	(**)
	bDriveDiagMessageAndNumber  : BOOL;
	m_GetDriveStatusState:INT;
	GetDriveStatusStateDone:BOOL;
	GetDriveStatusStateError:BOOL;
	GetDriveStatusTON: TON;
	//	
	fb_SoEReadDiagMessage_LeftTop: FB_SoEReadDiagMessage;
	fb_SoEReadDiagMessage_RightTop: FB_SoEReadDiagMessage;
	fb_SoEReadDiagMessage_LeftBottom: FB_SoEReadDiagMessage;
	fb_SoEReadDiagMessage_RightBottom: FB_SoEReadDiagMessage;
	DriveDiagMessage_LeftTop:STRING;
	DriveDiagMessage_RightTop:STRING;
	DriveDiagMessage_LeftBottom:STRING;
	DriveDiagMessage_RightBottom:STRING;
	fb_SoEReadDiagMessage_LeftIn: FB_SoEReadDiagMessage;
	fb_SoEReadDiagMessage_RightIn: FB_SoEReadDiagMessage;
	fb_SoEReadDiagMessage_LeftOut: FB_SoEReadDiagMessage;
	fb_SoEReadDiagMessage_RightOut: FB_SoEReadDiagMessage;
	DriveDiagMessage_LeftIn:STRING;
	DriveDiagMessage_RightIn:STRING;
	DriveDiagMessage_LeftOut:STRING;
	DriveDiagMessage_RightOut:STRING;
	//
	FB_SoEReadDiagNumber_LeftTop: FB_SoEReadDiagNumber;
	FB_SoEReadDiagNumber_RightTop: FB_SoEReadDiagNumber;
	FB_SoEReadDiagNumber_LeftBottom: FB_SoEReadDiagNumber;
	FB_SoEReadDiagNumber_RightBottom: FB_SoEReadDiagNumber;
	DriveDiagNumber_LeftTop:UDINT;
	DriveDiagNumber_RightTop:UDINT;
	DriveDiagNumber_LeftBottom:UDINT;
	DriveDiagNumber_RightBottom:UDINT;
	FB_SoEReadDiagNumber_LeftIn: FB_SoEReadDiagNumber;
	FB_SoEReadDiagNumber_RightIn: FB_SoEReadDiagNumber;
	FB_SoEReadDiagNumber_LeftOut: FB_SoEReadDiagNumber;
	FB_SoEReadDiagNumber_RightOut: FB_SoEReadDiagNumber;
	DriveDiagNumber_LeftIn:UDINT;
	DriveDiagNumber_RightIn:UDINT;
	DriveDiagNumber_LeftOut:UDINT;
	DriveDiagNumber_RightOut:UDINT;
	bReloadDriveDiagMessageAndNumber: BOOL;
	
	(*load IOC*)
	bExe_load_Prog: BOOL;
	NT_StartProcess_Load: NT_StartProcess;
	Exe_load_step: UINT;
	R_TRIG_ExeLoad: R_TRIG;
	Exe_Load_Done:BOOL;
	(*kill IOC*)
	bExe_Kill_Prog: BOOL;
	NT_StartProcess_Kill: NT_StartProcess;
	Exe_kill_step: UINT;
	R_TRIG_Exekill: R_TRIG;
	Exe_Kill_Done:BOOL;
	LoadOpcIocTON:TON;
	//
	IDControlReadyTon:TON;
	
	//
	//more parameters get:gear;feedback2 direction 
	//
	//GetMoreDriveStatus_FunctionON:BOOL:=TRUE;
	GetDriveStatusTON2: TON;
	//GearNumerator,st182
	st_p182_LeftTop:ST_P182;
	FB_SoERead_GearNumerator_LeftTop: FB_SoERead;
	st_p182_RightTop:ST_P182;
	FB_SoERead_GearNumerator_RightTop: FB_SoERead;
	st_p182_LeftBottom:ST_P182;
	FB_SoERead_GearNumerator_LeftBottom: FB_SoERead;
	st_p182_RightBottom:ST_P182;
	FB_SoERead_GearNumerator_RightBottom: FB_SoERead;
	GearNumeratorGet_LeftTop:UDINT;
	GearNumeratorGet_RightTop:UDINT;
	GearNumeratorGet_LeftBottom:UDINT;
	GearNumeratorGet_RightBottom:UDINT;
	GearNumeratorConfigured_LeftTop:UDINT;
	GearNumeratorConfigured_RightTop:UDINT;
	GearNumeratorConfigured_LeftBottom:UDINT;
	GearNumeratorConfigured_RightBottom:UDINT;
	st_p182_LeftIn:ST_P182;
	FB_SoERead_GearNumerator_LeftIn: FB_SoERead;
	st_p182_RightIn:ST_P182;
	FB_SoERead_GearNumerator_RightIn: FB_SoERead;
	st_p182_LeftOut:ST_P182;
	FB_SoERead_GearNumerator_LeftOut: FB_SoERead;
	st_p182_RightOut:ST_P182;
	FB_SoERead_GearNumerator_RightOut: FB_SoERead;
	GearNumeratorGet_LeftIn:UDINT;
	GearNumeratorGet_RightIn:UDINT;
	GearNumeratorGet_LeftOut:UDINT;
	GearNumeratorGet_RightOut:UDINT;
	GearNumeratorConfigured_LeftIn:UDINT;
	GearNumeratorConfigured_RightIn:UDINT;
	GearNumeratorConfigured_LeftOut:UDINT;
	GearNumeratorConfigured_RightOut:UDINT;
	//GearDenominator,st183
	st_p183_LeftTop:ST_P183;
	FB_SoERead_GearDenominator_LeftTop: FB_SoERead;
	st_p183_RightTop:ST_P183;
	FB_SoERead_GearDenominator_RightTop: FB_SoERead;
	st_p183_LeftBottom:ST_P183;
	FB_SoERead_GearDenominator_LeftBottom: FB_SoERead;
	st_p183_RightBottom:ST_P183;
	FB_SoERead_GearDenominator_RightBottom: FB_SoERead;
	GearDenominatorGet_LeftTop:UDINT;
	GearDenominatorGet_RightTop:UDINT;
	GearDenominatorGet_LeftBottom:UDINT;
	GearDenominatorGet_RightBottom:UDINT;
	GearDenominatorConfigured_LeftTop:UDINT;
	GearDenominatorConfigured_RightTop:UDINT;
	GearDenominatorConfigured_LeftBottom:UDINT;
	GearDenominatorConfigured_RightBottom:UDINT;
	st_p183_LeftIn:ST_P183;
	FB_SoERead_GearDenominator_LeftIn: FB_SoERead;
	st_p183_RightIn:ST_P183;
	FB_SoERead_GearDenominator_RightIn: FB_SoERead;
	st_p183_LeftOut:ST_P183;
	FB_SoERead_GearDenominator_LeftOut: FB_SoERead;
	st_p183_RightOut:ST_P183;
	FB_SoERead_GearDenominator_RightOut: FB_SoERead;
	GearDenominatorGet_LeftIn:UDINT;
	GearDenominatorGet_RightIn:UDINT;
	GearDenominatorGet_LeftOut:UDINT;
	GearDenominatorGet_RightOut:UDINT;
	GearDenominatorConfigured_LeftIn:UDINT;
	GearDenominatorConfigured_RightIn:UDINT;
	GearDenominatorConfigured_LeftOut:UDINT;
	GearDenominatorConfigured_RightOut:UDINT;
	//Feedback2direction,st180
	st_p180_LeftTop:ST_P180;
	FB_SoERead_Feedback2direction_LeftTop: FB_SoERead;
	st_p180_RightTop:ST_P180;
	FB_SoERead_Feedback2direction_RightTop: FB_SoERead;
	st_p180_LeftBottom:ST_P180;
	FB_SoERead_Feedback2direction_LeftBottom: FB_SoERead;
	st_p180_RightBottom:ST_P180;
	FB_SoERead_Feedback2direction_RightBottom: FB_SoERead;
	Feedback2directionGet_LeftTop:UINT;
	Feedback2directionGet_RightTop:UINT;
	Feedback2directionGet_LeftBottom:UINT;
	Feedback2directionGet_RightBottom:UINT;
	Feedback2directionConfigured_LeftTop:UINT;
	Feedback2directionConfigured_RightTop:UINT;
	Feedback2directionConfigured_LeftBottom:UINT;
	Feedback2directionConfigured_RightBottom:UINT;
	st_p180_LeftIn:ST_P180;
	FB_SoERead_Feedback2direction_LeftIn: FB_SoERead;
	st_p180_RightIn:ST_P180;
	FB_SoERead_Feedback2direction_RightIn: FB_SoERead;
	st_p180_LeftOut:ST_P180;
	FB_SoERead_Feedback2direction_LeftOut: FB_SoERead;
	st_p180_RightOut:ST_P180;
	FB_SoERead_Feedback2direction_RightOut: FB_SoERead;
	Feedback2directionGet_LeftIn:UINT;
	Feedback2directionGet_RightIn:UINT;
	Feedback2directionGet_LeftOut:UINT;
	Feedback2directionGet_RightOut:UINT;
	Feedback2directionConfigured_LeftIn:UINT;
	Feedback2directionConfigured_RightIn:UINT;
	Feedback2directionConfigured_LeftOut:UINT;
	Feedback2directionConfigured_RightOut:UINT;
	//
	//RestartDrivers
		(*重启驱动器*)
	btn_RestartDriversAll:BOOL;
	btn_RestartDriver1:BOOL;
	btn_RestartDriver2:BOOL;
	btn_RestartDriver3:BOOL;
	btn_RestartDriver4:BOOL;
	btn_RestartDriver5:BOOL;
	btn_RestartDriver6:BOOL;
	btn_RestartDriver7:BOOL;
	btn_RestartDriver8:BOOL;
	Relay_EL2624 AT %Q*:ARRAY[0..7]OF  BOOL;
	RestartDriver_RTRIG:R_TRIG;
	RestartDriver_TON:TON;
	RestartDriver_Triggered:BOOL;
	RestartDriver_State:DINT;
	RestartDriver_Done:BOOL;
	
	
	//
	//	LEHeartBeatMonitorFunction
	//
	LEHeartBeatMonitorFunctionOn: BOOL;
	LEHeartBeatFirstScan:BOOL;
	LEHeartBeatDeadZone : LREAL := 0; 
	LEHeartBeatAlarmTime : TIME := T#0.1S;
	
    //Pos_LeftTopLin_Last : LREAL; 
	Velo_LeftTopLin_Last : LREAL; 
	Pos_LeftTopMotor_Initial : LREAL; 
    StableTimer_LeftTopLin : TON; 
    StableTime_LeftTopLin : TIME; 
    DeltaVelo_LeftTopLin : LREAL; 
	IsInitialPositionSet_LeftTop: BOOL;
	MotorPosChange_LeftTop: LREAL;
	Threshold_LeftTopMotorPos:LREAL:=0.1;
	Threshold_LeftTopMotorVelo:LREAL:=0.2;
	Alarm_LeftTopLin:BOOL;
	Alarm_LeftTopMotorPos:BOOL;
	Alarm_LeftTopMotorVelo:BOOL;
	
	
	//Pos_RightTopLin_Last : LREAL; 
	Velo_RightTopLin_Last : LREAL; 
	Pos_RightTopMotor_Initial : LREAL; 
    StableTimer_RightTopLin : TON; 
    StableTime_RightTopLin : TIME; 
    DeltaVelo_RightTopLin : LREAL; 
	IsInitialPositionSet_RightTop: BOOL;
	MotorPosChange_RightTop: LREAL; 
	Threshold_RightTopMotorPos:LREAL:=0.1;
	Threshold_RightTopMotorVelo:LREAL:=0.2;
	Alarm_RightTopLin:BOOL;
	Alarm_RightTopMotorPos:BOOL;
	Alarm_RightTopMotorVelo:BOOL;
	
		
    //Pos_LeftBottomLin_Last : LREAL; 
	Velo_LeftBottomLin_Last : LREAL; 
	Pos_LeftBottomMotor_Initial : LREAL; 
    StableTimer_LeftBottomLin : TON; 
    StableTime_LeftBottomLin : TIME; 
    DeltaVelo_LeftBottomLin : LREAL; 
	IsInitialPositionSet_LeftBottom: BOOL;
	MotorPosChange_LeftBottom: LREAL; 
	Threshold_LeftBottomMotorPos:LREAL:=0.1;
	Threshold_LeftBottomMotorVelo:LREAL:=0.2;
	Alarm_LeftBottomLin:BOOL;
	Alarm_LeftBottomMotorPos:BOOL;
	Alarm_LeftBottomMotorVelo:BOOL;
	
	//Pos_RightBottomLin_Last : LREAL; 
	Velo_RightBottomLin_Last : LREAL; 
	Pos_RightBottomMotor_Initial : LREAL; 
    StableTimer_RightBottomLin : TON; 
    StableTime_RightBottomLin : TIME; 
    DeltaVelo_RightBottomLin : LREAL; 
	IsInitialPositionSet_RightBottom: BOOL;
	MotorPosChange_RightBottom: LREAL; 
	Threshold_RightBottomMotorPos:LREAL:=0.1;
	Threshold_RightBottomMotorVelo:LREAL:=0.2;
	Alarm_RightBottomLin:BOOL;
	Alarm_RightBottomMotorPos:BOOL;
	Alarm_RightBottomMotorVelo:BOOL;
	
	
    //Pos_LeftInLin_Last : LREAL; 
	Velo_LeftInLin_Last : LREAL; 
	Pos_LeftInMotor_Initial : LREAL; 
    StableTimer_LeftInLin : TON; 
    StableTime_LeftInLin : TIME; 
    DeltaVelo_LeftInLin : LREAL; 
	IsInitialPositionSet_LeftIn: BOOL;
	MotorPosChange_LeftIn: LREAL;
	Threshold_LeftInMotorPos:LREAL:=0.1;
	Threshold_LeftInMotorVelo:LREAL:=0.2;
	Alarm_LeftInLin:BOOL;
	Alarm_LeftInMotorPos:BOOL;
	Alarm_LeftInMotorVelo:BOOL;
	
	
	//Pos_RightInLin_Last : LREAL; 
	Velo_RightInLin_Last : LREAL; 
	Pos_RightInMotor_Initial : LREAL; 
    StableTimer_RightInLin : TON; 
    StableTime_RightInLin : TIME; 
    DeltaVelo_RightInLin : LREAL; 
	IsInitialPositionSet_RightIn: BOOL;
	MotorPosChange_RightIn: LREAL; 
	Threshold_RightInMotorPos:LREAL:=0.1;
	Threshold_RightInMotorVelo:LREAL:=0.2;
	Alarm_RightInLin:BOOL;
	Alarm_RightInMotorPos:BOOL;
	Alarm_RightInMotorVelo:BOOL;
	
		
    //Pos_LeftOutLin_Last : LREAL; 
	Velo_LeftOutLin_Last : LREAL; 
	Pos_LeftOutMotor_Initial : LREAL; 
    StableTimer_LeftOutLin : TON; 
    StableTime_LeftOutLin : TIME; 
    DeltaVelo_LeftOutLin : LREAL; 
	IsInitialPositionSet_LeftOut: BOOL;
	MotorPosChange_LeftOut: LREAL; 
	Threshold_LeftOutMotorPos:LREAL:=0.1;
	Threshold_LeftOutMotorVelo:LREAL:=0.2;
	Alarm_LeftOutLin:BOOL;
	Alarm_LeftOutMotorPos:BOOL;
	Alarm_LeftOutMotorVelo:BOOL;
	
	//Pos_RightOutLin_Last : LREAL; 
	Velo_RightOutLin_Last : LREAL; 
	Pos_RightOutMotor_Initial : LREAL; 
    StableTimer_RightOutLin : TON; 
    StableTime_RightOutLin : TIME; 
    DeltaVelo_RightOutLin : LREAL; 
	IsInitialPositionSet_RightOut: BOOL;
	MotorPosChange_RightOut: LREAL; 
	Threshold_RightOutMotorPos:LREAL:=0.1;
	Threshold_RightOutMotorVelo:LREAL:=0.2;
	Alarm_RightOutLin:BOOL;
	Alarm_RightOutMotorPos:BOOL;
	Alarm_RightOutMotorVelo:BOOL;
	//
	//fbMC_ReadParameter_ScaleFactor_LeftTopLIn: MC_ReadParameter;
	//fbMC_ReadParameter_ScaleFactor_RightTopLIn: MC_ReadParameter;
	//fbMC_ReadParameter_ScaleFactor_LeftBottomLIn: MC_ReadParameter;
	//fbMC_ReadParameter_ScaleFactor_RightBottomLIn: MC_ReadParameter;
	//ScaleFactor_LeftTopLin: LREAL;
	//ScaleFactor_RightTopLin: LREAL;
	//ScaleFactor_LeftBottomLin: LREAL;
	//ScaleFactor_RightBottomLin: LREAL;
	//
	//Velo_LeftTopMotor_DINT AT %I*: DINT;
	//Pos_LeftTopMotor_DINT AT %I*: DINT;
	//Velo_RightTopMotor_DINT AT %I*: DINT;
	//Pos_RightTopMotor_DINT AT %I*: DINT;
	//Velo_LeftBottomMotor_DINT AT %I*: DINT;
	//Pos_LeftBottomMotor_DINT AT %I*: DINT;
	//Velo_RightBottomMotor_DINT AT %I*: DINT;
	//Pos_RightBottomMotor_DINT AT %I*: DINT;
	
	(*setAxisPosition*)
	SetMotorAxisPosState: INT;
	FB_Set_MotorAxisPosition:FB_SetMotorAxisPosition;
	fb_ton4_2: TON;
	fb_ton5_2: TON;
	fb_ton6_2: TON;
	SetMotorAxisPositionDone: BOOL;
	
	btn_SetMotorAxisPosition: BOOL;
	MonitorMotorAndLEFunctionOn:BOOL:=TRUE;
END_VAR

(*加载Ricipe参数*)
A_InitRecipeParameters();
IF NOT loadParametersDone THEN
	RETURN;
END_IF
(*Restart TwinCAT*)
IF Global_Variables.m_restartTC THEN
(*首先关闭opcIocShell.exe*)	
	bExe_Kill_Prog:=TRUE;
	A_KillOpcIocShellExe();
(*重启TC*)
	IF Exe_Kill_Done THEN
		A_RestartTC();
	END_IF
END_IF
(*******InitAxisParameters*******)
A_InitAxisParameters();
(*******CheckLimitSwitch*******)
A_CheckLimitSwitch();
(*Check Kill Switch*)
A_CheckKillSwitch();
(*******PosDiff¼à¿Ø*******)
A_PosDiffDetectiion();
(*******³õÊ¼»¯SafePlc*******)
IF NOT simulation THEN
A_SafePlcStartInit();
END_IF
(************SetAxisPosition*********************)
IF  NOT USELinearEncoder AND setAxisPositionEnable AND btn_setAxisPosition THEN
	//IF NOT SerAxisPositionDone THEN
		FB_Set_AxisPosition.ValueSet_LeftTop:=ValueSet_LeftTop;
		FB_Set_AxisPosition.ValueSet_RightTop:=ValueSet_RightTop;
		FB_Set_AxisPosition.ValueSet_LeftBottom:=ValueSet_LeftBottom;
		FB_Set_AxisPosition.ValueSet_RightBottom:=ValueSet_RightBottom;
		FB_Set_AxisPosition.ValueSet_LeftIn:=ValueSet_LeftIn;
		FB_Set_AxisPosition.ValueSet_RightIn:=ValueSet_RightIn;
		FB_Set_AxisPosition.ValueSet_LeftOut:=ValueSet_LeftOut;
		FB_Set_AxisPosition.ValueSet_RightOut:=ValueSet_RightOut;
		A_SetAxisPosition();
	//END_IF
END_IF
(*******³Mode Select******)
IF SafePLCRunOK OR Simulation THEN
	IF pbSingleCarrierMode AND NOT pbDebugMode AND  NOT pbUserMode THEN
		SingleCarrierMode();
	ELSIF pbDebugMode AND NOT pbSingleCarrierMode AND NOT pbUserMode THEN
		DebugMode();
	ELSIF pbUserMode AND NOT pbSingleCarrierMode AND NOT pbDebugMode THEN
		UserMode();
	END_IF
END_IF
(*******Led Show******)
fb_led_Show();
(*******Check Power status******)
FB_Power(Check:=TRUE);
st_Power:=FB_Power.PowerState;

(*********RS232*********************)
BackgroundEL();
(*fbEL6001(TxBuffer:=TxBufferEL, RxBuffer:=RxBufferEL);*)

(*获取温度传感器数据*)
//A_GetTemperatureSensorsData();
(*低温补偿监控*)
//A_CryogenicCompensationMonitoring();

(*设置position bias*)
IF loadParametersDone AND (DriveStatus=1 OR simulation) THEN 
	A_SetLinearEncoderPositionBias();
END_IF
(*检查硬急停状态，包括安全限位、柜门急停、手持急停*)
A_CheckHardwareEmergencyStopStatus();
(*获取驱动器状态信息*)
IF NOT simulation THEN
	A_GetDriverStatus();
END_IF
(*IDControlReady*)
IF ((DriveStatus<>0 AND SafePLCRunOK) OR simulation) AND NOT Error THEN
	IDControlReady:=TRUE;
ELSE
	IDControlReady:=FALSE;
END_IF

(*IOC Start*)
//IF SafePLCRunOK OR simulation THEN
	bExe_load_Prog:=TRUE;
	A_LoadOpcIocShellExe();
//END_IF
(*检查光栅读数是否在范围内*)
A_CheckLinearEncoder();
(*RestartDrivers*)
A_RestartDrivers();


(*A_LEHeartBeatMonitor*)
IF LEHeartBeatMonitorFunctionOn THEN
	A_LEHeartBeatMonitor();
END_IF
(************SetMotorAxisPosition*********************)
//IDControl 1s after
fb_ton5_2.IN:=IDControlReady;
fb_ton5_2.PT:=T#1S;
fb_ton5_2();
IF fb_ton5_2.Q THEN
	btn_SetMotorAxisPosition:=TRUE;
END_IF
IF  USELinearEncoder AND btn_SetMotorAxisPosition THEN
	IF NOT SetMotorAxisPositionDone THEN
		FB_Set_MotorAxisPosition.ValueSet_LeftTop:=Pos_LeftTopLin;
		FB_Set_MotorAxisPosition.ValueSet_RightTop:=Pos_RightTopLin;
		FB_Set_MotorAxisPosition.ValueSet_LeftBottom:=Pos_LeftBottomLin;
		FB_Set_MotorAxisPosition.ValueSet_RightBottom:=Pos_RightBottomLin;
		FB_Set_MotorAxisPosition.ValueSet_LeftIn:=Pos_LeftInLin;
		FB_Set_MotorAxisPosition.ValueSet_RightIn:=Pos_RightInLin;
		FB_Set_MotorAxisPosition.ValueSet_LeftOut:=Pos_LeftOutLin;
		FB_Set_MotorAxisPosition.ValueSet_RightOut:=Pos_RightOutLin;
		A_SetMotorAxisPosition();
	END_IF
END_IF
(*A_MonitorMotorAndLE*)
IF MonitorMotorAndLEFunctionOn AND SetMotorAxisPositionDone THEN
	A_MonitorMotorAndLE();
END_IF
(*A_CheckMaxVelocity*)
A_CheckMaxVelocity();

ACTION A_CheckHardwareEmergencyStopStatus:
IF 	NOT KS_LeftTop_Far_Contact1 OR
	NOT KS_LeftTop_Far_Contact2 OR
	NOT KS_RightTop_Far_Contact1 OR
	NOT KS_RightTop_Far_Contact2 OR
	NOT KS_LeftBottom_Far_Contact1 OR
	NOT KS_LeftBottom_Far_Contact2 OR
	NOT KS_RightBottom_Far_Contact1 OR
	NOT KS_RightBottom_Far_Contact2 OR
	
	NOT KS_LeftTop_Near_Contact1 OR
	NOT KS_LeftTop_Near_Contact2 OR
	NOT KS_RightTop_Near_Contact1 OR
	NOT KS_RightTop_Near_Contact2 OR
	NOT KS_LeftBottom_Near_Contact1 OR
	NOT KS_LeftBottom_Near_Contact2 OR
	NOT KS_RightBottom_Near_Contact1 OR
	NOT KS_RightBottom_Near_Contact2 OR
	
	NOT KS_LeftIn_Far_Contact1 OR
	NOT KS_LeftIn_Far_Contact2 OR
	NOT KS_RightIn_Far_Contact1 OR
	NOT KS_RightIn_Far_Contact2 OR
	NOT KS_LeftOut_Far_Contact1 OR
	NOT KS_LeftOut_Far_Contact2 OR
	NOT KS_RightOut_Far_Contact1 OR
	NOT KS_RightOut_Far_Contact2 OR
	
	NOT KS_LeftIn_Near_Contact1 OR
	NOT KS_LeftIn_Near_Contact2 OR
	NOT KS_RightIn_Near_Contact1 OR
	NOT KS_RightIn_Near_Contact2 OR
	NOT KS_LeftOut_Near_Contact1 OR
	NOT KS_LeftOut_Near_Contact2 OR
	NOT KS_RightOut_Near_Contact1 OR
	NOT KS_RightOut_Near_Contact2 OR
(*E-STOP*)
	NOT KS_CabinetEmergency_contact1 OR
	NOT KS_CabinetEmergency_contact2 OR
	NOT KS_handEmergency1_Contact1 OR
	NOT KS_handEmergency1_Contact2 OR
	NOT KS_handEmergency2_Contact1 OR
	NOT KS_handEmergency2_Contact2 OR
	NOT KS_softEmergency2_Contact THEN
	Hardware_EmergencyStop:=FALSE;
ELSE
	Hardware_EmergencyStop:=TRUE;
END_IF
END_ACTION

ACTION A_CheckKillSwitch:
IF simulation THEN
	KS_LeftTop_Far_Contact1:=TRUE;
	KS_LeftTop_Far_Contact2:=TRUE;
	KS_LeftTop_Near_Contact1:=TRUE;
	KS_LeftTop_Near_Contact2:=TRUE;
	KS_RightTop_Far_Contact1:=TRUE;
	KS_RightTop_Far_Contact2:=TRUE;
	KS_RightTop_Near_Contact1:=TRUE;
	KS_RightTop_Near_Contact2:=TRUE;
	KS_LeftBottom_Far_Contact1:=TRUE;
	KS_LeftBottom_Far_Contact2:=TRUE;
	KS_LeftBottom_Near_Contact1:=TRUE;
	KS_LeftBottom_Near_Contact2:=TRUE;	
	KS_RightBottom_Far_Contact1:=TRUE;
	KS_RightBottom_Far_Contact2:=TRUE;
	KS_RightBottom_Near_Contact1:=TRUE;
	KS_RightBottom_Near_Contact2:=TRUE;	

	KS_LeftIn_Far_Contact1:=TRUE;
	KS_LeftIn_Far_Contact2:=TRUE;
	KS_LeftIn_Near_Contact1:=TRUE;
	KS_LeftIn_Near_Contact2:=TRUE;
	KS_RightIn_Far_Contact1:=TRUE;
	KS_RightIn_Far_Contact2:=TRUE;
	KS_RightIn_Near_Contact1:=TRUE;
	KS_RightIn_Near_Contact2:=TRUE;
	KS_LeftOut_Far_Contact1:=TRUE;
	KS_LeftOut_Far_Contact2:=TRUE;
	KS_LeftOut_Near_Contact1:=TRUE;
	KS_LeftOut_Near_Contact2:=TRUE;	
	KS_RightOut_Far_Contact1:=TRUE;
	KS_RightOut_Far_Contact2:=TRUE;
	KS_RightOut_Near_Contact1:=TRUE;
	KS_RightOut_Near_Contact2:=TRUE;		
	(*E-STOP*)
	KS_CabinetEmergency_contact1:=TRUE;
	KS_CabinetEmergency_contact2:=TRUE;	
	KS_handEmergency1_Contact1:=TRUE;
	KS_handEmergency1_Contact2:=TRUE;
	KS_handEmergency2_Contact1:=TRUE;
	KS_handEmergency2_Contact2:=TRUE;
	
	KS_softEmergency2_Contact:=TRUE;

ELSE
	KS_LeftTop_Near_Contact1:=EL1904[1];//c3
	KS_LeftTop_Near_Contact2:=EL1904[2];//c4
	KS_LeftTop_Far_Contact1:=EL1904[3];//c1
	KS_LeftTop_Far_Contact2:=EL1904[4];//c2

	KS_RightTop_Near_Contact1:=EL1904[5];
	KS_RightTop_Near_Contact2:=EL1904[6];
	KS_RightTop_Far_Contact1:=EL1904[7];
	KS_RightTop_Far_Contact2:=EL1904[8];

	KS_LeftBottom_Near_Contact1:=EL1904[9];
	KS_LeftBottom_Near_Contact2:=EL1904[10];
	KS_LeftBottom_Far_Contact1:=EL1904[11];
	KS_LeftBottom_Far_Contact2:=EL1904[12];

	KS_RightBottom_Near_Contact1:=EL1904[13];
	KS_RightBottom_Near_Contact2:=EL1904[14];	
	KS_RightBottom_Far_Contact1:=EL1904[15];
	KS_RightBottom_Far_Contact2:=EL1904[16];
	
	KS_LeftIn_Near_Contact1:=EL1904[17];//c3
	KS_LeftIn_Near_Contact2:=EL1904[18];//c4
	KS_LeftIn_Far_Contact1:=EL1904[19];//c1
	KS_LeftIn_Far_Contact2:=EL1904[20];//c2

	KS_RightIn_Near_Contact1:=EL1904[21];
	KS_RightIn_Near_Contact2:=EL1904[22];
	KS_RightIn_Far_Contact1:=EL1904[23];
	KS_RightIn_Far_Contact2:=EL1904[24];

	KS_LeftOut_Near_Contact1:=EL1904[25];
	KS_LeftOut_Near_Contact2:=EL1904[26];
	KS_LeftOut_Far_Contact1:=EL1904[27];
	KS_LeftOut_Far_Contact2:=EL1904[28];

	KS_RightOut_Near_Contact1:=EL1904[29];
	KS_RightOut_Near_Contact2:=EL1904[30];	
	KS_RightOut_Far_Contact1:=EL1904[31];
	KS_RightOut_Far_Contact2:=EL1904[32];
	
	(*E-STOP*)
	KS_CabinetEmergency_contact1:=EL1904[33];
	KS_CabinetEmergency_contact2:=EL1904[34];
	
	KS_handEmergency1_Contact1:=EL1904[35];
	KS_handEmergency1_Contact2:=EL1904[36];
	KS_handEmergency2_Contact1:=EL1904[37];
	KS_handEmergency2_Contact2:=EL1904[38];
	
	KS_softEmergency2_Contact:=EL1904[39];
	END_IF
END_ACTION

ACTION A_CheckLimitSwitch:
(**)
IF simulation THEN
	(**)
	LS_LeftTop_Far:=TRUE;
	LS_LeftTop_Near:=TRUE;
	LS_RightTop_Far:=TRUE;
	LS_RightTop_Near:=TRUE;
	LS_LeftBottom_Far:=TRUE;
	LS_LeftBottom_Near:=TRUE;
	LS_RightBottom_Far:=TRUE;
	LS_RightBottom_Near:=TRUE;	
	LS_LeftIn_Far:=TRUE;
	LS_LeftIn_Near:=TRUE;
	LS_RightIn_Far:=TRUE;
	LS_RightIn_Near:=TRUE;
	LS_LeftOut_Far:=TRUE;
	LS_LeftOut_Near:=TRUE;
	LS_RightOut_Far:=TRUE;
	LS_RightOut_Near:=TRUE;
ELSE
	LS_LeftTop_Near :=el1808_D1[1];
	LS_LeftTop_Far:=el1808_D1[2];
	LS_RightTop_Near:=el1808_D1[3];
	LS_RightTop_Far:=el1808_D1[4];
	LS_LeftBottom_Near:=el1808_D1[5];
	LS_LeftBottom_Far:=el1808_D1[6];
	LS_RightBottom_Near:=el1808_D1[7];
	LS_RightBottom_Far:=el1808_D1[8];
	LS_LeftIn_Near :=el1808_D1[9];
	LS_LeftIn_Far:=el1808_D1[10];
	LS_RightIn_Near:=el1808_D1[11];
	LS_RightIn_Far:=el1808_D1[12];
	LS_LeftOut_Near:=el1808_D1[13];
	LS_LeftOut_Far:=el1808_D1[14];
	LS_RightOut_Near:=el1808_D1[15];
	LS_RightOut_Far:=el1808_D1[16];
END_IF

(********************)
Unreach_LS_Far:=LS_LeftTop_Far AND LS_RightTop_Far AND LS_LeftBottom_Far AND LS_RightBottom_Far
				AND LS_LeftIn_Far AND LS_RightIn_Far AND LS_LeftOut_Far AND LS_RightOut_Far;
Unreach_LS_Near:=LS_LeftTop_Near AND LS_RightTop_Near AND LS_LeftBottom_Near AND LS_RightBottom_Near
				AND LS_LeftIn_Near AND LS_RightIn_Near AND LS_LeftOut_Near AND LS_RightOut_Near;
END_ACTION

ACTION A_CheckLinearEncoder:
//LEProtectionPosition
min_UserLEProtectionGapPosition:=min_UserGapPositionNew-min_ThresholdGapSoft2LEProtection;//回程误差有0.1mm
max_UserLEProtectionGapPosition:=max_UserGapPositionNew+max_ThresholdGapSoft2LEProtection;
//如果没有使用光栅、或者光栅参数没设置好，则不检查光栅位置
IF NOT USELinearEncoder OR NOT PositionBiasDone THEN
	RETURN;
END_IF
IF Pos_LeftTopLin <=0 THEN
	ErrorID:=1101;
	Error:=TRUE;
	ErrorDescription:='Pos_LeftTopLin <=0';
	FB_PlcEmergencyStop();
	LED_Error:=TRUE;
END_IF
IF Pos_RightTopLin <=0 THEN
	ErrorID:=1102;
	Error:=TRUE;
	ErrorDescription:='Pos_RightTopLin <=0';
	FB_PlcEmergencyStop();
	LED_Error:=TRUE;
END_IF
IF Pos_LeftBottomLin <=0 THEN
	ErrorID:=1103;
	Error:=TRUE;
	ErrorDescription:='Pos_LeftBottomLin <=0';
	FB_PlcEmergencyStop();
	LED_Error:=TRUE;
END_IF
IF Pos_RightBottomLin <=0 THEN
	ErrorID:=1104;
	Error:=TRUE;
	ErrorDescription:='Pos_RightBottomLin <=0';
	FB_PlcEmergencyStop();
	LED_Error:=TRUE;
END_IF
//
IF Pos_LeftInLin <=0 THEN
	ErrorID:=1105;
	Error:=TRUE;
	ErrorDescription:='Pos_LeftInLin <=0';
	FB_PlcEmergencyStop();
	LED_Error:=TRUE;
END_IF
IF Pos_RightInLin <=0 THEN
	ErrorID:=1106;
	Error:=TRUE;
	ErrorDescription:='Pos_RightInLin <=0';
	FB_PlcEmergencyStop();
	LED_Error:=TRUE;
END_IF
IF Pos_LeftOutLin <=0 THEN
	ErrorID:=1107;
	Error:=TRUE;
	ErrorDescription:='Pos_LeftOutLin <=0';
	FB_PlcEmergencyStop();
	LED_Error:=TRUE;
END_IF
IF Pos_RightOutLin <=0 THEN
	ErrorID:=1108;
	Error:=TRUE;
	ErrorDescription:='Pos_RightOutLin <=0';
	FB_PlcEmergencyStop();
	LED_Error:=TRUE;
END_IF
//
//Gap方向
//
//
IF Pos_LeftTopLin >max_UserLEProtectionGapPosition/2 THEN
	ErrorID:=1105;
	Error:=TRUE;
	ErrorDescription:='Pos_LeftTopLin >max_UserLEProtectionGapPosition/2';
	FB_PlcEmergencyStop();
	LED_Error:=TRUE;
END_IF
IF Pos_RightTopLin >max_UserLEProtectionGapPosition/2 THEN
	ErrorID:=1106;
	Error:=TRUE;
	ErrorDescription:='Pos_RightTopLin>max_UserLEProtectionGapPosition/2';
	FB_PlcEmergencyStop();
	LED_Error:=TRUE;
END_IF
IF Pos_LeftBottomLin >max_UserLEProtectionGapPosition/2 THEN
	ErrorID:=1107;
	Error:=TRUE;
	ErrorDescription:='Pos_LeftBottomLin >max_UserLEProtectionGapPosition/2';
	FB_PlcEmergencyStop();
	LED_Error:=TRUE;
END_IF
IF Pos_RightBottomLin >max_UserLEProtectionGapPosition/2 THEN
	ErrorID:=1108;
	Error:=TRUE;
	ErrorDescription:='Pos_RightBottomLin >max_UserLEProtectionGapPosition/2';
	FB_PlcEmergencyStop();
	LED_Error:=TRUE;
END_IF
IF Pos_LeftInLin >max_UserLEProtectionGapPosition/2 THEN
	ErrorID:=1105;
	Error:=TRUE;
	ErrorDescription:='Pos_LeftInLin >max_UserLEProtectionGapPosition/2';
	FB_PlcEmergencyStop();
	LED_Error:=TRUE;
END_IF
IF Pos_RightInLin >max_UserLEProtectionGapPosition/2 THEN
	ErrorID:=1106;
	Error:=TRUE;
	ErrorDescription:='Pos_RightInLin>max_UserLEProtectionGapPosition/2';
	FB_PlcEmergencyStop();
	LED_Error:=TRUE;
END_IF
IF Pos_LeftOutLin >max_UserLEProtectionGapPosition/2 THEN
	ErrorID:=1107;
	Error:=TRUE;
	ErrorDescription:='Pos_LeftOutLin >max_UserLEProtectionGapPosition/2';
	FB_PlcEmergencyStop();
	LED_Error:=TRUE;
END_IF
IF Pos_RightOutLin >max_UserLEProtectionGapPosition/2 THEN
	ErrorID:=1108;
	Error:=TRUE;
	ErrorDescription:='Pos_RightOutLin >max_UserLEProtectionGapPosition/2';
	FB_PlcEmergencyStop();
	LED_Error:=TRUE;
END_IF
//
IF Pos_LeftTopLin <min_UserLEProtectionGapPosition/2 THEN
	ErrorID:=1109;
	Error:=TRUE;
	ErrorDescription:='Pos_LeftTopLin <min_UserLEProtectionGapPosition/2';
	FB_PlcEmergencyStop();
	LED_Error:=TRUE;
END_IF
IF Pos_RightTopLin <min_UserLEProtectionGapPosition/2 THEN
	ErrorID:=1110;
	Error:=TRUE;
	ErrorDescription:='Pos_RightTopLin<min_UserLEProtectionGapPosition/2';
	FB_PlcEmergencyStop();
	LED_Error:=TRUE;
END_IF
IF Pos_LeftBottomLin <min_UserLEProtectionGapPosition/2 THEN
	ErrorID:=1111;
	Error:=TRUE;
	ErrorDescription:='Pos_LeftBottomLin <min_UserLEProtectionGapPosition';
	FB_PlcEmergencyStop();
	LED_Error:=TRUE;
END_IF
IF Pos_RightBottomLin <min_UserLEProtectionGapPosition/2 THEN
	ErrorID:=1112;
	Error:=TRUE;
	ErrorDescription:='Pos_RightBottomLin <min_UserLEProtectionGapPosition';
	FB_PlcEmergencyStop();
	LED_Error:=TRUE;
END_IF
IF Pos_LeftInLin <min_UserLEProtectionGapPosition/2 THEN
	ErrorID:=1109;
	Error:=TRUE;
	ErrorDescription:='Pos_LeftInLin <min_UserLEProtectionGapPosition/2';
	FB_PlcEmergencyStop();
	LED_Error:=TRUE;
END_IF
IF Pos_RightInLin <min_UserLEProtectionGapPosition/2 THEN
	ErrorID:=1110;
	Error:=TRUE;
	ErrorDescription:='Pos_RightInLin<min_UserLEProtectionGapPosition/2';
	FB_PlcEmergencyStop();
	LED_Error:=TRUE;
END_IF
IF Pos_LeftOutLin <min_UserLEProtectionGapPosition/2 THEN
	ErrorID:=1111;
	Error:=TRUE;
	ErrorDescription:='Pos_LeftOutLin <min_UserLEProtectionGapPosition';
	FB_PlcEmergencyStop();
	LED_Error:=TRUE;
END_IF
IF Pos_RightOutLin <min_UserLEProtectionGapPosition/2 THEN
	ErrorID:=1112;
	Error:=TRUE;
	ErrorDescription:='Pos_RightOutLin <min_UserLEProtectionGapPosition';
	FB_PlcEmergencyStop();
	LED_Error:=TRUE;
END_IF
END_ACTION

ACTION A_CheckMaxVelocity:
IF NOT USELinearEncoder OR NOT PositionBiasDone OR NOT IDControlReady THEN
	RETURN;
END_IF
IF NOT st_Power THEN
	RETURN;
END_IF
//Monitoring Motor and LE Position/Velocity
MaxVelocityGlobalVelocity:=MAX(max_UserGapVelocityNew,max_UserTaperVelocityNew,UserMode.max_SS_StepVelocity,
							UserMode.Global_ChainProtection_MPS_MoveVelocity
	,UserMode.Global_ChainProtection_EPS_MoveVelocity);
IF 	ABS(Velo_LeftTopLin) > MaxVelocityGlobalVelocity*1.1/2 THEN
	ErrorID:=7001;
	Error:=TRUE;
	ErrorDescription:='ABS(Velo_LeftTopLin) > MaxVelocityGlobalVelocity*1.1/2';
	FB_PlcEmergencyStop();
	LED_Error:=TRUE;
END_IF
IF 	ABS(Velo_LeftTopMotor) > MaxVelocityGlobalVelocity*1.1/2 THEN
	ErrorID:=7002;
	Error:=TRUE;
	ErrorDescription:='ABS(Velo_LeftTopMotor) > MaxVelocityGlobalVelocity*1.1/2';
	FB_PlcEmergencyStop();
	LED_Error:=TRUE;
END_IF
IF 	ABS(Velo_RightTopLin) > MaxVelocityGlobalVelocity*1.1/2 THEN
	ErrorID:=7003;
	Error:=TRUE;
	ErrorDescription:='ABS(Velo_RightTopLin) > MaxVelocityGlobalVelocity*1.1/2';
	FB_PlcEmergencyStop();
	LED_Error:=TRUE;
END_IF
IF 	ABS(Velo_RightTopMotor) > MaxVelocityGlobalVelocity*1.1/2 THEN
	ErrorID:=7004;
	Error:=TRUE;
	ErrorDescription:='ABS(Velo_RightTopMotor) > MaxVelocityGlobalVelocity*1.1/2';
	FB_PlcEmergencyStop();
	LED_Error:=TRUE;
END_IF
IF 	ABS(Velo_LeftBottomLin) > MaxVelocityGlobalVelocity*1.1/2 THEN
	ErrorID:=7005;
	Error:=TRUE;
	ErrorDescription:='ABS(Velo_LeftBottomLin) > MaxVelocityGlobalVelocity*1.1/2';
	FB_PlcEmergencyStop();
	LED_Error:=TRUE;
END_IF
IF 	ABS(Velo_LeftBottomMotor) > MaxVelocityGlobalVelocity*1.1/2 THEN
	ErrorID:=7006;
	Error:=TRUE;
	ErrorDescription:='ABS(Velo_LeftBottomMotor) > MaxVelocityGlobalVelocity*1.1/2';
	FB_PlcEmergencyStop();
	LED_Error:=TRUE;
END_IF
IF 	ABS(Velo_RightBottomLin) > MaxVelocityGlobalVelocity*1.1/2 THEN
	ErrorID:=7007;
	Error:=TRUE;
	ErrorDescription:='ABS(Velo_RightBottomLin) > MaxVelocityGlobalVelocity*1.1/2';
	FB_PlcEmergencyStop();
	LED_Error:=TRUE;
END_IF
IF 	ABS(Velo_RightBottomMotor) > MaxVelocityGlobalVelocity*1.1/2 THEN
	ErrorID:=7008;
	Error:=TRUE;
	ErrorDescription:='ABS(Velo_RighBottomMotor) > MaxVelocityGlobalVelocity*1.1/2';
	FB_PlcEmergencyStop();
	LED_Error:=TRUE;
END_IF

IF 	ABS(Velo_LeftInLin) > MaxVelocityGlobalVelocity*1.1/2 THEN
	ErrorID:=7009;
	Error:=TRUE;
	ErrorDescription:='ABS(Velo_LeftInLin) > MaxVelocityGlobalVelocity*1.1/2';
	FB_PlcEmergencyStop();
	LED_Error:=TRUE;
END_IF
IF 	ABS(Velo_LeftInMotor) > MaxVelocityGlobalVelocity*1.1/2 THEN
	ErrorID:=7010;
	Error:=TRUE;
	ErrorDescription:='ABS(Velo_LeftInMotor) > MaxVelocityGlobalVelocity*1.1/2';
	FB_PlcEmergencyStop();
	LED_Error:=TRUE;
END_IF
IF 	ABS(Velo_RightInLin) > MaxVelocityGlobalVelocity*1.1/2 THEN
	ErrorID:=7011;
	Error:=TRUE;
	ErrorDescription:='ABS(Velo_RightInLin) > MaxVelocityGlobalVelocity*1.1/2';
	FB_PlcEmergencyStop();
	LED_Error:=TRUE;
END_IF
IF 	ABS(Velo_RightInMotor) > MaxVelocityGlobalVelocity*1.1/2 THEN
	ErrorID:=7012;
	Error:=TRUE;
	ErrorDescription:='ABS(Velo_RightInMotor) > MaxVelocityGlobalVelocity*1.1/2';
	FB_PlcEmergencyStop();
	LED_Error:=TRUE;
END_IF
IF 	ABS(Velo_LeftOutLin) > MaxVelocityGlobalVelocity*1.1/2 THEN
	ErrorID:=7013;
	Error:=TRUE;
	ErrorDescription:='ABS(Velo_LeftOutLin) > MaxVelocityGlobalVelocity*1.1/2';
	FB_PlcEmergencyStop();
	LED_Error:=TRUE;
END_IF
IF 	ABS(Velo_LeftOutMotor) > MaxVelocityGlobalVelocity*1.1/2 THEN
	ErrorID:=7014;
	Error:=TRUE;
	ErrorDescription:='ABS(Velo_LeftOutMotor) > MaxVelocityGlobalVelocity*1.1/2';
	FB_PlcEmergencyStop();
	LED_Error:=TRUE;
END_IF
IF 	ABS(Velo_RightOutLin) > MaxVelocityGlobalVelocity*1.1/2 THEN
	ErrorID:=7015;
	Error:=TRUE;
	ErrorDescription:='ABS(Velo_RightOutLin) > MaxVelocityGlobalVelocity*1.1/2';
	FB_PlcEmergencyStop();
	LED_Error:=TRUE;
END_IF
IF 	ABS(Velo_RightOutMotor) > MaxVelocityGlobalVelocity*1.1/2 THEN
	ErrorID:=7016;
	Error:=TRUE;
	ErrorDescription:='ABS(Velo_RighOutMotor) > MaxVelocityGlobalVelocity*1.1/2';
	FB_PlcEmergencyStop();
	LED_Error:=TRUE;
END_IF
END_ACTION

ACTION A_CryogenicCompensationMonitoring:
//没有传感器OR不是CPMU不低温补偿OR低温不到位，均不补偿
IF NOT HasTemperatureSensorOrNot OR NOT CryogenicCompensationOn THEN //OR temperatureStatus<>2 THEN
	//不补偿
	CryogenicCompensation_LeftTop:=0;
	CryogenicCompensation_RightTop:=0;
	CryogenicCompensation_LeftBottom:=0;
	CryogenicCompensation_RightBottom:=0;
ELSE
	CryogenicCompensationConditionsReady:=TRUE;//条件具备，可以低温补偿
	//检查补偿值，单轴补偿范围均在0-1内
	IF CryogenicCompensation_LeftTop>1 OR CryogenicCompensation_LeftTop<=0 THEN
			Error:=TRUE;
			ErrorID:=1201;
			ErrorDescription:='CryogenicCompensation_LeftTop>1 OR CryogenicCompensation_LeftTop<=0';
			FB_PlcEmergencyStop();
	END_IF
	IF CryogenicCompensation_RightTop>1 OR CryogenicCompensation_RightTop<=0 THEN
			Error:=TRUE;
			ErrorID:=1202;
			ErrorDescription:='CryogenicCompensation_RightTop>1 OR CryogenicCompensation_RightTop<=0';
			FB_PlcEmergencyStop();
	END_IF
	IF CryogenicCompensation_LeftBottom>1 OR CryogenicCompensation_LeftBottom<=0 THEN
			Error:=TRUE;
			ErrorID:=1203;
			ErrorDescription:='CryogenicCompensation_LeftBottom>1 OR CryogenicCompensation_LeftBottom<=0';
			FB_PlcEmergencyStop();
	END_IF
	IF CryogenicCompensation_RightBottom>1 OR CryogenicCompensation_RightBottom<=0 THEN
			Error:=TRUE;
			ErrorID:=1204;
			ErrorDescription:='CryogenicCompensation_RightBottom>1 OR CryogenicCompensation_RightBottom<=0';
			FB_PlcEmergencyStop();
	END_IF
END_IF
//若在低温补偿模式，但是温度没到低温区间，则Emergency，不允许启动
(*
IF CryogenicCompensationOn AND temperatureStatus<>2 THEN
			Error:=TRUE;
			ErrorID:=1205;
			ErrorDescription:='CryogenicCompensationOn AND temperatureStatus<>2';
			FB_PlcEmergencyStop();
END_IF
*)
END_ACTION

ACTION A_GetDriverStatus:
//
//DriveMessage/Drive Number/Gear number/feedback2 direction
//
IF bReloadDriveDiagMessageAndNumber THEN
	m_GetDriveStatusState:=0;
	bReloadDriveDiagMessageAndNumber:=FALSE;
END_IF
GetDriveStatusTON(PT:=T#1S);
GetDriveStatusTON2(PT:=T#0.1S);
A_GetDriverStatusMC();
CASE m_GetDriveStatusState OF
	0:
		GetDriveStatusTON.IN:=TRUE;
		m_GetDriveStatusState:=1;
	1:
		IF GetDriveStatusTON.Q THEN
			bDriveDiagMessageAndNumber:=TRUE;
			m_GetDriveStatusState:=2;
		END_IF
	2:
		GetDriveStatusTON.IN:=FALSE;
		DriveDiagMessage_LeftTop:=fb_SoEReadDiagMessage_LeftTop.sDiagMessage.strData;
		DriveDiagMessage_RightTop:=fb_SoEReadDiagMessage_RightTop.sDiagMessage.strData;
		DriveDiagMessage_LeftBottom:=fb_SoEReadDiagMessage_LeftBottom.sDiagMessage.strData;
		DriveDiagMessage_RightBottom:=fb_SoEReadDiagMessage_RightBottom.sDiagMessage.strData;
		DriveDiagMessage_LeftIn:=fb_SoEReadDiagMessage_LeftIn.sDiagMessage.strData;
		DriveDiagMessage_RightIn:=fb_SoEReadDiagMessage_RightIn.sDiagMessage.strData;
		DriveDiagMessage_LeftOut:=fb_SoEReadDiagMessage_LeftOut.sDiagMessage.strData;
		DriveDiagMessage_RightOut:=fb_SoEReadDiagMessage_RightOut.sDiagMessage.strData;
		//
		DriveDiagNumber_LeftTop:=FB_SoEReadDiagNumber_LeftTop.iDiagNumber;
		DriveDiagNumber_RightTop:=FB_SoEReadDiagNumber_RightTop.iDiagNumber;
		DriveDiagNumber_LeftBottom:=FB_SoEReadDiagNumber_LeftBottom.iDiagNumber;
		DriveDiagNumber_RightBottom:=FB_SoEReadDiagNumber_RightBottom.iDiagNumber;
		DriveDiagNumber_LeftIn:=FB_SoEReadDiagNumber_LeftIn.iDiagNumber;
		DriveDiagNumber_RightIn:=FB_SoEReadDiagNumber_RightIn.iDiagNumber;
		DriveDiagNumber_LeftOut:=FB_SoEReadDiagNumber_LeftOut.iDiagNumber;
		DriveDiagNumber_RightOut:=FB_SoEReadDiagNumber_RightOut.iDiagNumber;
		//
		GearNumeratorGet_LeftTop:=st_p182_LeftTop.Feedback_2_geat_numerator;
		GearNumeratorGet_RightTop:=st_p182_RightTop.Feedback_2_geat_numerator;
		GearNumeratorGet_LeftBottom:=st_p182_LeftBottom.Feedback_2_geat_numerator;
		GearNumeratorGet_RightBottom:=st_p182_RightBottom.Feedback_2_geat_numerator;
		GearNumeratorGet_LeftIn:=st_p182_LeftIn.Feedback_2_geat_numerator;
		GearNumeratorGet_RightIn:=st_p182_RightIn.Feedback_2_geat_numerator;
		GearNumeratorGet_LeftOut:=st_p182_LeftOut.Feedback_2_geat_numerator;
		GearNumeratorGet_RightOut:=st_p182_RightOut.Feedback_2_geat_numerator;
		//
		GearDenominatorGet_LeftTop:=st_p183_LeftTop.Feedback_2_geat_denominator;
		GearDenominatorGet_RightTop:=st_p183_RightTop.Feedback_2_geat_denominator;
		GearDenominatorGet_LeftBottom:=st_p183_LeftBottom.Feedback_2_geat_denominator;
		GearDenominatorGet_RightBottom:=st_p183_RightBottom.Feedback_2_geat_denominator;
		GearDenominatorGet_LeftIn:=st_p183_LeftIn.Feedback_2_geat_denominator;
		GearDenominatorGet_RightIn:=st_p183_RightIn.Feedback_2_geat_denominator;
		GearDenominatorGet_LeftOut:=st_p183_LeftOut.Feedback_2_geat_denominator;
		GearDenominatorGet_RightOut:=st_p183_RightOut.Feedback_2_geat_denominator;
		//
		Feedback2directionGet_LeftTop:=st_p180_LeftTop.Feedback_direction;
		Feedback2directionGet_RightTop:=st_p180_RightTop.Feedback_direction;
		Feedback2directionGet_LeftBottom:=st_p180_LeftBottom.Feedback_direction;
		Feedback2directionGet_RightBottom:=st_p180_RightBottom.Feedback_direction;
		Feedback2directionGet_LeftIn:=st_p180_LeftIn.Feedback_direction;
		Feedback2directionGet_RightIn:=st_p180_RightIn.Feedback_direction;
		Feedback2directionGet_LeftOut:=st_p180_LeftOut.Feedback_direction;
		Feedback2directionGet_RightOut:=st_p180_RightOut.Feedback_direction;
		//
		IF 	NOT FB_SoEReadDiagMessage_LeftTop.bBusy
			AND NOT FB_SoEReadDiagMessage_RightTop.bBusy
			AND NOT FB_SoEReadDiagMessage_LeftBottom.bBusy
			AND NOT FB_SoEReadDiagMessage_RightBottom.bBusy 
			AND NOT FB_SoEReadDiagNumber_LeftTop.bBusy
			AND NOT FB_SoEReadDiagNumber_RightTop.bBusy
			AND NOT FB_SoEReadDiagNumber_LeftBottom.bBusy
			AND NOT FB_SoEReadDiagNumber_RightBottom.bBusy 
			AND NOT FB_SoERead_GearNumerator_LeftTop.bBusy 
			AND NOT FB_SoERead_GearNumerator_RightTop.bBusy 
			AND NOT FB_SoERead_GearNumerator_LeftBottom.bBusy 
			AND NOT FB_SoERead_GearNumerator_RightBottom.bBusy 
			AND NOT FB_SoERead_GearDenominator_LeftTop.bBusy 
			AND NOT FB_SoERead_GearDenominator_RightTop.bBusy 
			AND NOT FB_SoERead_GearDenominator_LeftBottom.bBusy 
			AND NOT FB_SoERead_GearDenominator_RightBottom.bBusy 
			AND NOT FB_SoERead_Feedback2direction_LeftTop.bBusy 
			AND NOT FB_SoERead_Feedback2direction_RightTop.bBusy 
			AND NOT FB_SoERead_Feedback2direction_LeftBottom.bBusy 
			AND NOT FB_SoERead_Feedback2direction_RightBottom.bBusy	
			AND NOT FB_SoEReadDiagMessage_LeftIn.bBusy
			AND NOT FB_SoEReadDiagMessage_RightIn.bBusy
			AND NOT FB_SoEReadDiagMessage_LeftOut.bBusy
			AND NOT FB_SoEReadDiagMessage_RightOut.bBusy 
			AND NOT FB_SoEReadDiagNumber_LeftIn.bBusy
			AND NOT FB_SoEReadDiagNumber_RightIn.bBusy
			AND NOT FB_SoEReadDiagNumber_LeftOut.bBusy
			AND NOT FB_SoEReadDiagNumber_RightOut.bBusy 
			AND NOT FB_SoERead_GearNumerator_LeftIn.bBusy 
			AND NOT FB_SoERead_GearNumerator_RightIn.bBusy 
			AND NOT FB_SoERead_GearNumerator_LeftOut.bBusy 
			AND NOT FB_SoERead_GearNumerator_RightOut.bBusy 
			AND NOT FB_SoERead_GearDenominator_LeftIn.bBusy 
			AND NOT FB_SoERead_GearDenominator_RightIn.bBusy 
			AND NOT FB_SoERead_GearDenominator_LeftOut.bBusy 
			AND NOT FB_SoERead_GearDenominator_RightOut.bBusy 
			AND NOT FB_SoERead_Feedback2direction_LeftIn.bBusy 
			AND NOT FB_SoERead_Feedback2direction_RightIn.bBusy 
			AND NOT FB_SoERead_Feedback2direction_LeftOut.bBusy 
			AND NOT FB_SoERead_Feedback2direction_RightOut.bBusy	THEN
				GetDriveStatusTON2.IN:=TRUE;
				IF GetDriveStatusTON2.Q THEN
					m_GetDriveStatusState:=88;
				END_IF
		END_IF
		IF 	FB_SoEReadDiagMessage_LeftTop.bError
			OR FB_SoEReadDiagMessage_RightTop.bError
			OR FB_SoEReadDiagMessage_LeftBottom.bError
			OR FB_SoEReadDiagMessage_RightBottom.bError
			OR FB_SoEReadDiagNumber_LeftTop.bError
			OR FB_SoEReadDiagNumber_RightTop.bError
			OR FB_SoEReadDiagNumber_LeftBottom.bError
			OR FB_SoEReadDiagNumber_RightBottom.bError 
			OR FB_SoERead_GearNumerator_LeftTop.bError 
			OR FB_SoERead_GearNumerator_RightTop.bError 
			OR FB_SoERead_GearNumerator_LeftBottom.bError 
			OR FB_SoERead_GearNumerator_RightBottom.bError 
			OR FB_SoERead_GearDenominator_LeftTop.bError 
			OR FB_SoERead_GearDenominator_RightTop.bError 
			OR FB_SoERead_GearDenominator_LeftBottom.bError 
			OR FB_SoERead_GearDenominator_RightBottom.bError 
			OR FB_SoERead_Feedback2direction_LeftTop.bError 
			OR FB_SoERead_Feedback2direction_RightTop.bError 
			OR FB_SoERead_Feedback2direction_LeftBottom.bError 
			OR FB_SoERead_Feedback2direction_RightBottom.bError 
			OR FB_SoEReadDiagMessage_LeftIn.bError
			OR fb_SoEReadDiagMessage_RightIn.bError
			OR fb_SoEReadDiagMessage_LeftOut.bError
			OR fb_SoEReadDiagMessage_RightOut.bError
			OR FB_SoEReadDiagNumber_LeftIn.bError
			OR FB_SoEReadDiagNumber_RightIn.bError
			OR FB_SoEReadDiagNumber_LeftOut.bError
			OR FB_SoEReadDiagNumber_RightOut.bError 
			OR FB_SoERead_GearNumerator_LeftIn.bError 
			OR FB_SoERead_GearNumerator_RightIn.bError 
			OR FB_SoERead_GearNumerator_LeftOut.bError 
			OR FB_SoERead_GearNumerator_RightOut.bError 
			OR FB_SoERead_GearDenominator_LeftIn.bError 
			OR FB_SoERead_GearDenominator_RightIn.bError 
			OR FB_SoERead_GearDenominator_LeftOut.bError 
			OR FB_SoERead_GearDenominator_RightOut.bError 
			OR FB_SoERead_Feedback2direction_LeftIn.bError 
			OR FB_SoERead_Feedback2direction_RightIn.bError 
			OR FB_SoERead_Feedback2direction_LeftOut.bError 
			OR FB_SoERead_Feedback2direction_RightOut.bError 
		THEN
			m_GetDriveStatusState:=-100;
		END_IF
		
	88:
		bDriveDiagMessageAndNumber:=FALSE;
		A_GetDriverStatusMC();
		GetDriveStatusStateDone:=TRUE;
		GetDriveStatusStateError:=FALSE;
		//
		(*Drive Status*)
		//D012, Axis state machine: Control and power section ready,53266
		IF DriveDiagNumber_LeftTop=16#D012 AND DriveDiagNumber_RightTop=16#D012
			AND DriveDiagNumber_LeftBottom=16#D012 AND DriveDiagNumber_RightBottom=16#D012 
			AND DriveDiagNumber_LeftIn=16#D012 AND DriveDiagNumber_RightIn=16#D012
			AND DriveDiagNumber_LeftOut=16#D012 AND DriveDiagNumber_RightOut=16#D012 THEN
			DriveStatus:=1;
		//D013, Axis state machine: Axis in operation,53267
		ELSIF DriveDiagNumber_LeftTop=16#D013 AND DriveDiagNumber_RightTop=16#D013
			AND DriveDiagNumber_LeftBottom=16#D013 AND DriveDiagNumber_RightBottom=16#D013 
			AND DriveDiagNumber_LeftIn=16#D013 AND DriveDiagNumber_RightIn=16#D013
			AND DriveDiagNumber_LeftOut=16#D013 AND DriveDiagNumber_RightOut=16#D013THEN
			DriveStatus:=2;
		//D014，Axis state machine: Axis halt.53266和53267中间会经历这么一个状态，算正常状态
		ELSIF DriveDiagNumber_LeftTop=16#D014 AND DriveDiagNumber_RightTop=16#D014
			AND DriveDiagNumber_LeftBottom=16#D014 AND DriveDiagNumber_RightBottom=16#D014 
			AND DriveDiagNumber_LeftIn=16#D014 AND DriveDiagNumber_RightIn=16#D014
			AND DriveDiagNumber_LeftOut=16#D014 AND DriveDiagNumber_RightOut=16#D014 THEN
			DriveStatus:=3;
		ELSE
			DriveStatus:=0;
		END_IF
		//
		//
		//	//check statusGet and status configured
		IF 	GearNumeratorGet_LeftTop<>GearNumeratorConfigured_LeftTop 
			OR GearNumeratorGet_RightTop<>GearNumeratorConfigured_RightTop
			OR GearNumeratorGet_LeftBottom<>GearNumeratorConfigured_LeftBottom 
			OR GearNumeratorGet_RightBottom<>GearNumeratorConfigured_RightBottom
			OR GearDenominatorGet_LeftTop<>GearDenominatorConfigured_LeftTop 
			OR GearDenominatorGet_RightTop<>GearDenominatorConfigured_RightTop
			OR GearDenominatorGet_LeftBottom<>GearDenominatorConfigured_LeftBottom 
			OR GearDenominatorGet_RightBottom<>GearDenominatorConfigured_RightBottom
			OR GearNumeratorGet_LeftIn<>GearNumeratorConfigured_LeftIn 
			OR GearNumeratorGet_RightIn<>GearNumeratorConfigured_RightIn
			OR GearNumeratorGet_LeftOut<>GearNumeratorConfigured_LeftOut 
			OR GearNumeratorGet_RightOut<>GearNumeratorConfigured_RightOut
			OR GearDenominatorGet_LeftIn<>GearDenominatorConfigured_LeftIn 
			OR GearDenominatorGet_RightIn<>GearDenominatorConfigured_RightIn
			OR GearDenominatorGet_LeftOut<>GearDenominatorConfigured_LeftOut 
			OR GearDenominatorGet_RightOut<>GearDenominatorConfigured_RightOut THEN 
				bDriveDiagMessageAndNumber:=FALSE;
				A_GetDriverStatusMC();
				GetDriveStatusStateDone:=FALSE;
				GetDriveStatusStateError:=TRUE;
				Error:=TRUE;
				ErrorId:=1302;
				ErrorDescription:='gear Parameters Error';
				Plc_EmergencyStop:=FALSE;
		END_IF
		IF USELinearEncoder THEN
			IF 	Feedback2directionGet_LeftTop<>Feedback2directionConfigured_LeftTop 
				OR Feedback2directionGet_RightTop<>Feedback2directionConfigured_RightTop
				OR Feedback2directionGet_LeftBottom<>Feedback2directionConfigured_LeftBottom 
				OR Feedback2directionGet_RightBottom<Feedback2directionConfigured_RightBottom 
				OR Feedback2directionGet_LeftIn<>Feedback2directionConfigured_LeftIn 
				OR Feedback2directionGet_RightIn<>Feedback2directionConfigured_RightIn
				OR Feedback2directionGet_LeftOut<>Feedback2directionConfigured_LeftOut 
				OR Feedback2directionGet_RightOut<Feedback2directionConfigured_RightOut THEN
					bDriveDiagMessageAndNumber:=FALSE;
					A_GetDriverStatusMC();
					GetDriveStatusStateDone:=FALSE;
					GetDriveStatusStateError:=TRUE;
					Error:=TRUE;
					ErrorId:=1303;
					ErrorDescription:='fb2direction Error';
					Plc_EmergencyStop:=FALSE;	
			END_IF
		END_IF
		m_GetDriveStatusState:=0;
	-100:
		bDriveDiagMessageAndNumber:=FALSE;
		A_GetDriverStatusMC();
		GetDriveStatusStateDone:=FALSE;
		GetDriveStatusStateError:=TRUE;
		Error:=TRUE;
		ErrorId:=1301;
		ErrorDescription:='GetDriveStatusStateError';
END_CASE
END_ACTION

ACTION A_GetDriverStatusMC:
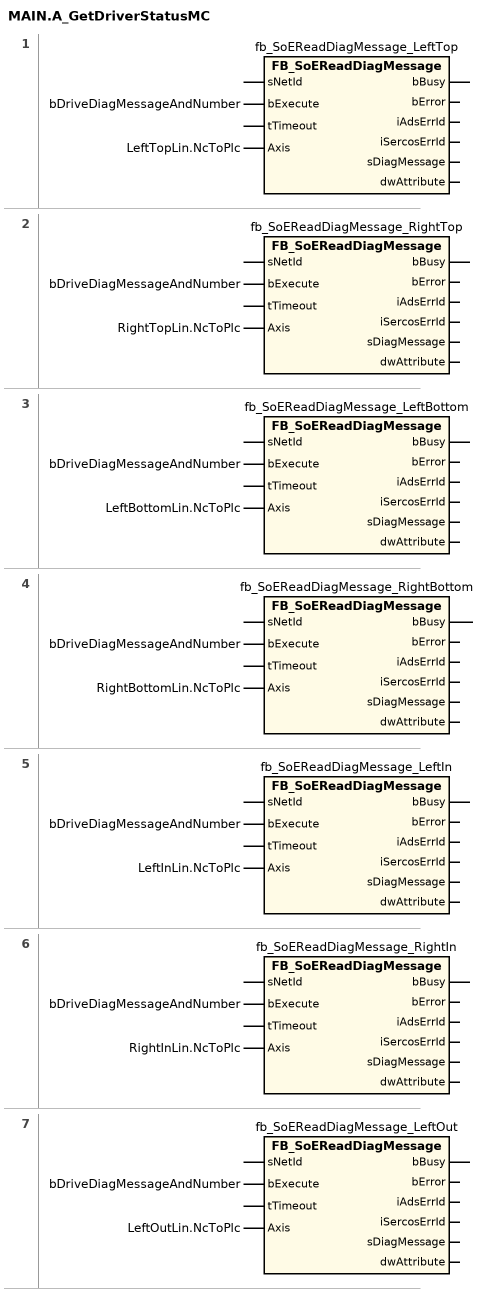
// NETWORK 1
fb_SoEReadDiagMessage_LeftTop(bExecute := bDriveDiagMessageAndNumber, Axis := LeftTopLin.NcToPlc); // FB_SoEReadDiagMessage

// NETWORK 2
fb_SoEReadDiagMessage_RightTop(bExecute := bDriveDiagMessageAndNumber, Axis := RightTopLin.NcToPlc); // FB_SoEReadDiagMessage

// NETWORK 3
fb_SoEReadDiagMessage_LeftBottom(bExecute := bDriveDiagMessageAndNumber, Axis := LeftBottomLin.NcToPlc); // FB_SoEReadDiagMessage

// NETWORK 4
fb_SoEReadDiagMessage_RightBottom(bExecute := bDriveDiagMessageAndNumber, Axis := RightBottomLin.NcToPlc); // FB_SoEReadDiagMessage

// NETWORK 5
fb_SoEReadDiagMessage_LeftIn(bExecute := bDriveDiagMessageAndNumber, Axis := LeftInLin.NcToPlc); // FB_SoEReadDiagMessage

// NETWORK 6
fb_SoEReadDiagMessage_RightIn(bExecute := bDriveDiagMessageAndNumber, Axis := RightInLin.NcToPlc); // FB_SoEReadDiagMessage

// NETWORK 7
fb_SoEReadDiagMessage_LeftOut(bExecute := bDriveDiagMessageAndNumber, Axis := LeftOutLin.NcToPlc); // FB_SoEReadDiagMessage

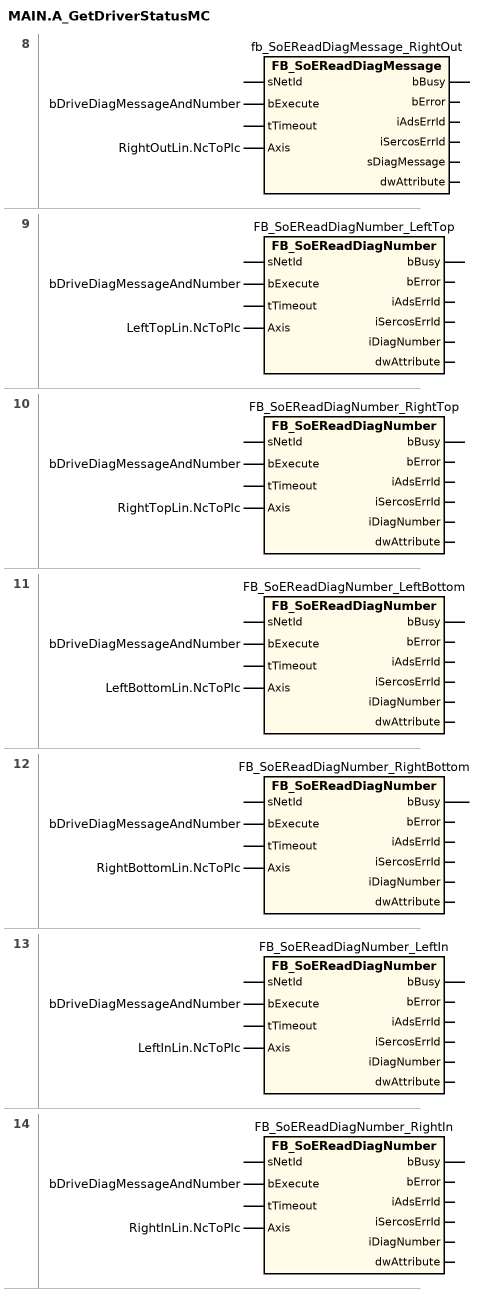
// NETWORK 8
fb_SoEReadDiagMessage_RightOut(bExecute := bDriveDiagMessageAndNumber, Axis := RightOutLin.NcToPlc); // FB_SoEReadDiagMessage

// NETWORK 9
FB_SoEReadDiagNumber_LeftTop(bExecute := bDriveDiagMessageAndNumber, Axis := LeftTopLin.NcToPlc); // FB_SoEReadDiagNumber

// NETWORK 10
FB_SoEReadDiagNumber_RightTop(bExecute := bDriveDiagMessageAndNumber, Axis := RightTopLin.NcToPlc); // FB_SoEReadDiagNumber

// NETWORK 11
FB_SoEReadDiagNumber_LeftBottom(bExecute := bDriveDiagMessageAndNumber, Axis := LeftBottomLin.NcToPlc); // FB_SoEReadDiagNumber

// NETWORK 12
FB_SoEReadDiagNumber_RightBottom(bExecute := bDriveDiagMessageAndNumber, Axis := RightBottomLin.NcToPlc); // FB_SoEReadDiagNumber

// NETWORK 13
FB_SoEReadDiagNumber_LeftIn(bExecute := bDriveDiagMessageAndNumber, Axis := LeftInLin.NcToPlc); // FB_SoEReadDiagNumber

// NETWORK 14
FB_SoEReadDiagNumber_RightIn(bExecute := bDriveDiagMessageAndNumber, Axis := RightInLin.NcToPlc); // FB_SoEReadDiagNumber

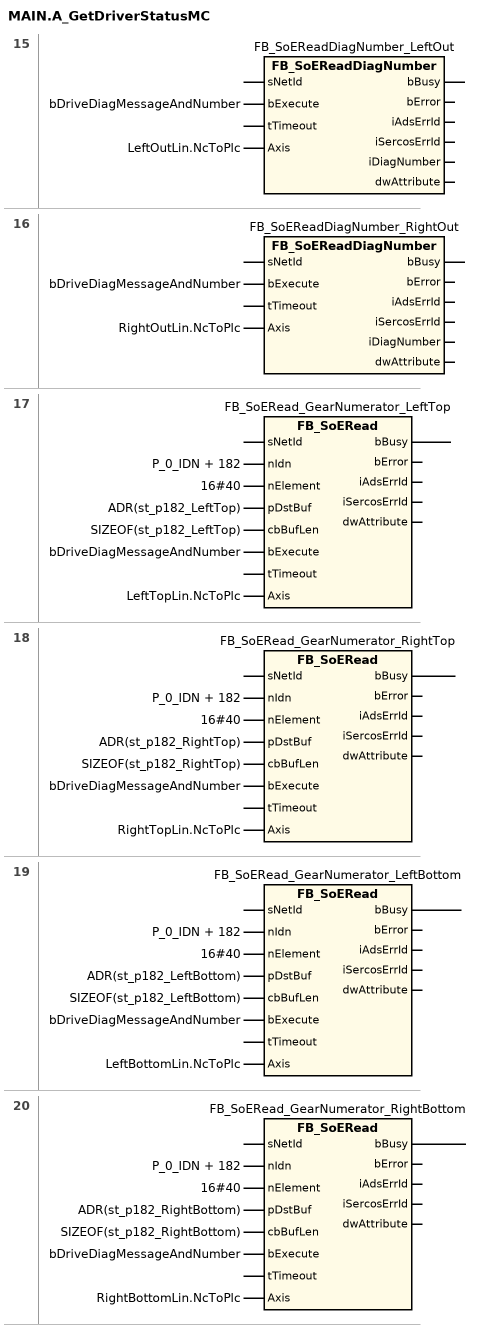
// NETWORK 15
FB_SoEReadDiagNumber_LeftOut(bExecute := bDriveDiagMessageAndNumber, Axis := LeftOutLin.NcToPlc); // FB_SoEReadDiagNumber

// NETWORK 16
FB_SoEReadDiagNumber_RightOut(bExecute := bDriveDiagMessageAndNumber, Axis := RightOutLin.NcToPlc); // FB_SoEReadDiagNumber

// NETWORK 17
FB_SoERead_GearNumerator_LeftTop(
    nIdn := P_0_IDN + 182,
    nElement := 16#40,
    pDstBuf := ADR(st_p182_LeftTop),
    cbBufLen := SIZEOF(st_p182_LeftTop),
    bExecute := bDriveDiagMessageAndNumber,
    Axis := LeftTopLin.NcToPlc); // FB_SoERead

// NETWORK 18
FB_SoERead_GearNumerator_RightTop(
    nIdn := P_0_IDN + 182,
    nElement := 16#40,
    pDstBuf := ADR(st_p182_RightTop),
    cbBufLen := SIZEOF(st_p182_RightTop),
    bExecute := bDriveDiagMessageAndNumber,
    Axis := RightTopLin.NcToPlc); // FB_SoERead

// NETWORK 19
FB_SoERead_GearNumerator_LeftBottom(
    nIdn := P_0_IDN + 182,
    nElement := 16#40,
    pDstBuf := ADR(st_p182_LeftBottom),
    cbBufLen := SIZEOF(st_p182_LeftBottom),
    bExecute := bDriveDiagMessageAndNumber,
    Axis := LeftBottomLin.NcToPlc); // FB_SoERead

// NETWORK 20
FB_SoERead_GearNumerator_RightBottom(
    nIdn := P_0_IDN + 182,
    nElement := 16#40,
    pDstBuf := ADR(st_p182_RightBottom),
    cbBufLen := SIZEOF(st_p182_RightBottom),
    bExecute := bDriveDiagMessageAndNumber,
    Axis := RightBottomLin.NcToPlc); // FB_SoERead

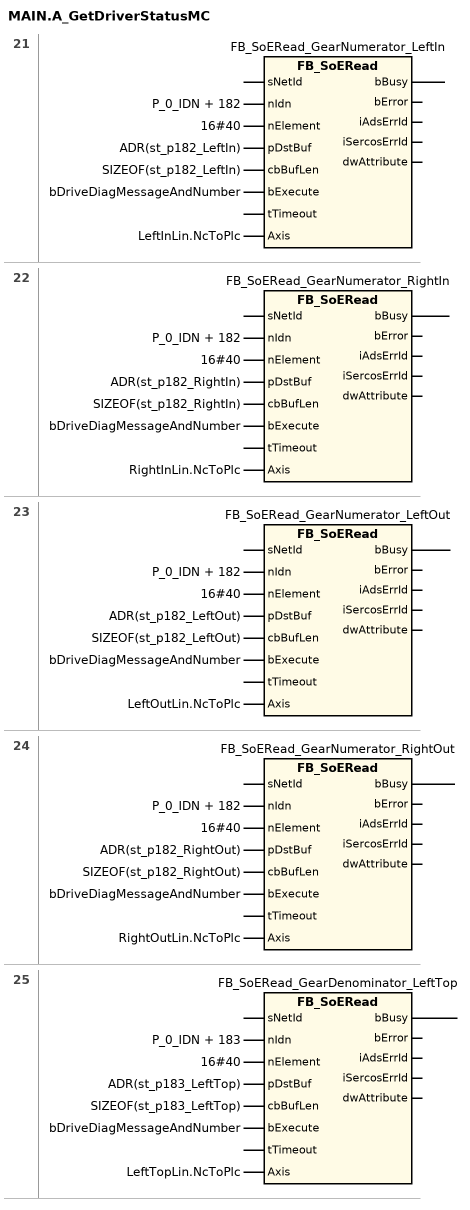
// NETWORK 21
FB_SoERead_GearNumerator_LeftIn(
    nIdn := P_0_IDN + 182,
    nElement := 16#40,
    pDstBuf := ADR(st_p182_LeftIn),
    cbBufLen := SIZEOF(st_p182_LeftIn),
    bExecute := bDriveDiagMessageAndNumber,
    Axis := LeftInLin.NcToPlc); // FB_SoERead

// NETWORK 22
FB_SoERead_GearNumerator_RightIn(
    nIdn := P_0_IDN + 182,
    nElement := 16#40,
    pDstBuf := ADR(st_p182_RightIn),
    cbBufLen := SIZEOF(st_p182_RightIn),
    bExecute := bDriveDiagMessageAndNumber,
    Axis := RightInLin.NcToPlc); // FB_SoERead

// NETWORK 23
FB_SoERead_GearNumerator_LeftOut(
    nIdn := P_0_IDN + 182,
    nElement := 16#40,
    pDstBuf := ADR(st_p182_LeftOut),
    cbBufLen := SIZEOF(st_p182_LeftOut),
    bExecute := bDriveDiagMessageAndNumber,
    Axis := LeftOutLin.NcToPlc); // FB_SoERead

// NETWORK 24
FB_SoERead_GearNumerator_RightOut(
    nIdn := P_0_IDN + 182,
    nElement := 16#40,
    pDstBuf := ADR(st_p182_RightOut),
    cbBufLen := SIZEOF(st_p182_RightOut),
    bExecute := bDriveDiagMessageAndNumber,
    Axis := RightOutLin.NcToPlc); // FB_SoERead

// NETWORK 25
FB_SoERead_GearDenominator_LeftTop(
    nIdn := P_0_IDN + 183,
    nElement := 16#40,
    pDstBuf := ADR(st_p183_LeftTop),
    cbBufLen := SIZEOF(st_p183_LeftTop),
    bExecute := bDriveDiagMessageAndNumber,
    Axis := LeftTopLin.NcToPlc); // FB_SoERead

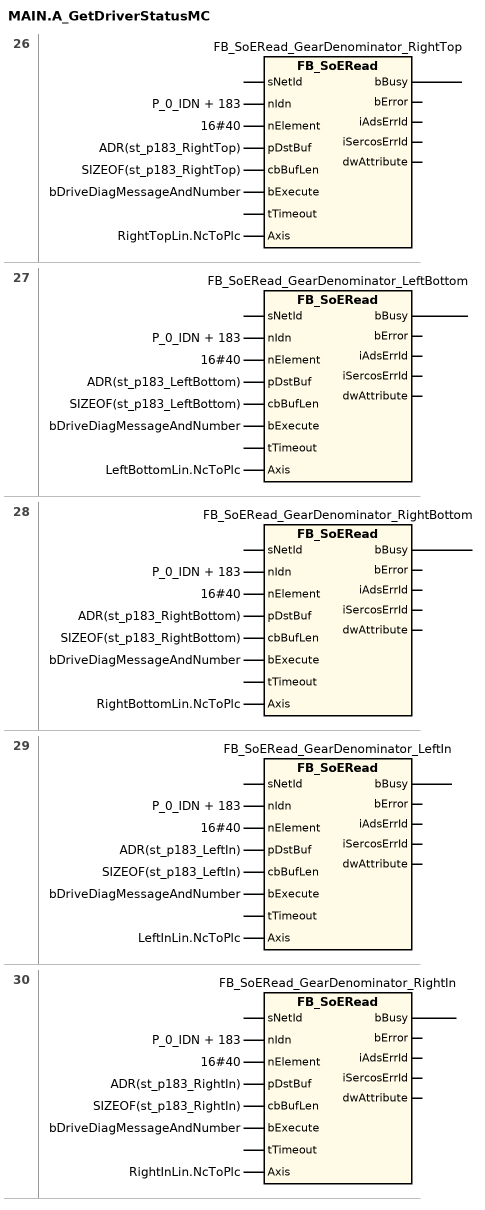
// NETWORK 26
FB_SoERead_GearDenominator_RightTop(
    nIdn := P_0_IDN + 183,
    nElement := 16#40,
    pDstBuf := ADR(st_p183_RightTop),
    cbBufLen := SIZEOF(st_p183_RightTop),
    bExecute := bDriveDiagMessageAndNumber,
    Axis := RightTopLin.NcToPlc); // FB_SoERead

// NETWORK 27
FB_SoERead_GearDenominator_LeftBottom(
    nIdn := P_0_IDN + 183,
    nElement := 16#40,
    pDstBuf := ADR(st_p183_LeftBottom),
    cbBufLen := SIZEOF(st_p183_LeftBottom),
    bExecute := bDriveDiagMessageAndNumber,
    Axis := LeftBottomLin.NcToPlc); // FB_SoERead

// NETWORK 28
FB_SoERead_GearDenominator_RightBottom(
    nIdn := P_0_IDN + 183,
    nElement := 16#40,
    pDstBuf := ADR(st_p183_RightBottom),
    cbBufLen := SIZEOF(st_p183_RightBottom),
    bExecute := bDriveDiagMessageAndNumber,
    Axis := RightBottomLin.NcToPlc); // FB_SoERead

// NETWORK 29
FB_SoERead_GearDenominator_LeftIn(
    nIdn := P_0_IDN + 183,
    nElement := 16#40,
    pDstBuf := ADR(st_p183_LeftIn),
    cbBufLen := SIZEOF(st_p183_LeftIn),
    bExecute := bDriveDiagMessageAndNumber,
    Axis := LeftInLin.NcToPlc); // FB_SoERead

// NETWORK 30
FB_SoERead_GearDenominator_RightIn(
    nIdn := P_0_IDN + 183,
    nElement := 16#40,
    pDstBuf := ADR(st_p183_RightIn),
    cbBufLen := SIZEOF(st_p183_RightIn),
    bExecute := bDriveDiagMessageAndNumber,
    Axis := RightInLin.NcToPlc); // FB_SoERead

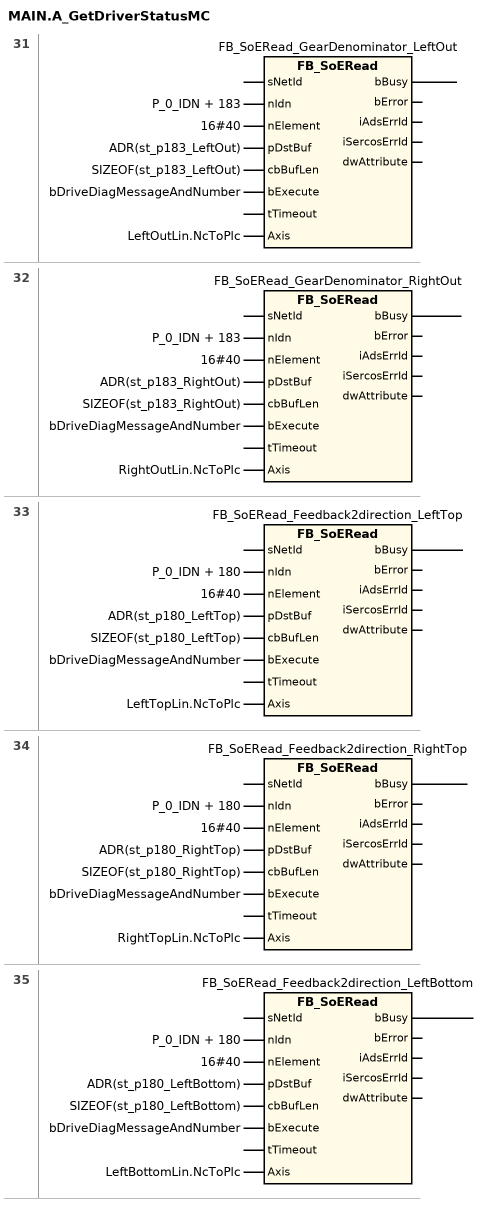
// NETWORK 31
FB_SoERead_GearDenominator_LeftOut(
    nIdn := P_0_IDN + 183,
    nElement := 16#40,
    pDstBuf := ADR(st_p183_LeftOut),
    cbBufLen := SIZEOF(st_p183_LeftOut),
    bExecute := bDriveDiagMessageAndNumber,
    Axis := LeftOutLin.NcToPlc); // FB_SoERead

// NETWORK 32
FB_SoERead_GearDenominator_RightOut(
    nIdn := P_0_IDN + 183,
    nElement := 16#40,
    pDstBuf := ADR(st_p183_RightOut),
    cbBufLen := SIZEOF(st_p183_RightOut),
    bExecute := bDriveDiagMessageAndNumber,
    Axis := RightOutLin.NcToPlc); // FB_SoERead

// NETWORK 33
FB_SoERead_Feedback2direction_LeftTop(
    nIdn := P_0_IDN + 180,
    nElement := 16#40,
    pDstBuf := ADR(st_p180_LeftTop),
    cbBufLen := SIZEOF(st_p180_LeftTop),
    bExecute := bDriveDiagMessageAndNumber,
    Axis := LeftTopLin.NcToPlc); // FB_SoERead

// NETWORK 34
FB_SoERead_Feedback2direction_RightTop(
    nIdn := P_0_IDN + 180,
    nElement := 16#40,
    pDstBuf := ADR(st_p180_RightTop),
    cbBufLen := SIZEOF(st_p180_RightTop),
    bExecute := bDriveDiagMessageAndNumber,
    Axis := RightTopLin.NcToPlc); // FB_SoERead

// NETWORK 35
FB_SoERead_Feedback2direction_LeftBottom(
    nIdn := P_0_IDN + 180,
    nElement := 16#40,
    pDstBuf := ADR(st_p180_LeftBottom),
    cbBufLen := SIZEOF(st_p180_LeftBottom),
    bExecute := bDriveDiagMessageAndNumber,
    Axis := LeftBottomLin.NcToPlc); // FB_SoERead

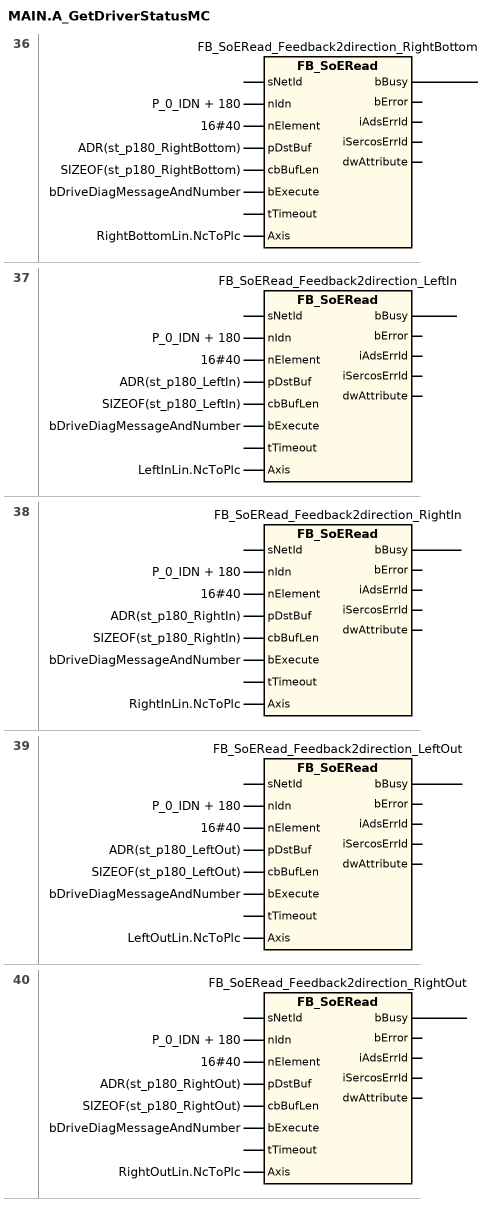
// NETWORK 36
FB_SoERead_Feedback2direction_RightBottom(
    nIdn := P_0_IDN + 180,
    nElement := 16#40,
    pDstBuf := ADR(st_p180_RightBottom),
    cbBufLen := SIZEOF(st_p180_RightBottom),
    bExecute := bDriveDiagMessageAndNumber,
    Axis := RightBottomLin.NcToPlc); // FB_SoERead

// NETWORK 37
FB_SoERead_Feedback2direction_LeftIn(
    nIdn := P_0_IDN + 180,
    nElement := 16#40,
    pDstBuf := ADR(st_p180_LeftIn),
    cbBufLen := SIZEOF(st_p180_LeftIn),
    bExecute := bDriveDiagMessageAndNumber,
    Axis := LeftInLin.NcToPlc); // FB_SoERead

// NETWORK 38
FB_SoERead_Feedback2direction_RightIn(
    nIdn := P_0_IDN + 180,
    nElement := 16#40,
    pDstBuf := ADR(st_p180_RightIn),
    cbBufLen := SIZEOF(st_p180_RightIn),
    bExecute := bDriveDiagMessageAndNumber,
    Axis := RightInLin.NcToPlc); // FB_SoERead

// NETWORK 39
FB_SoERead_Feedback2direction_LeftOut(
    nIdn := P_0_IDN + 180,
    nElement := 16#40,
    pDstBuf := ADR(st_p180_LeftOut),
    cbBufLen := SIZEOF(st_p180_LeftOut),
    bExecute := bDriveDiagMessageAndNumber,
    Axis := LeftOutLin.NcToPlc); // FB_SoERead

// NETWORK 40
FB_SoERead_Feedback2direction_RightOut(
    nIdn := P_0_IDN + 180,
    nElement := 16#40,
    pDstBuf := ADR(st_p180_RightOut),
    cbBufLen := SIZEOF(st_p180_RightOut),
    bExecute := bDriveDiagMessageAndNumber,
    Axis := RightOutLin.NcToPlc); // FB_SoERead
END_ACTION

ACTION A_GetTemperatureSensorsData:
//sensor_1
dut_sensor_datas_1.data_byte[3]:=Sensor_Reading_1[0];
dut_sensor_datas_1.data_byte[2]:=Sensor_Reading_1[1];
dut_sensor_datas_1.data_byte[1]:=Sensor_Reading_1[2];
dut_sensor_datas_1.data_byte[0]:=Sensor_Reading_1[3];
TemperatureSensors_1:=DINT_TO_LREAL(LREAL_TO_DINT(dut_sensor_datas_1.data_lreal*100))/100;
//sensor_2
dut_sensor_datas_2.data_byte[3]:=Sensor_Reading_2[0];
dut_sensor_datas_2.data_byte[2]:=Sensor_Reading_2[1];
dut_sensor_datas_2.data_byte[1]:=Sensor_Reading_2[2];
dut_sensor_datas_2.data_byte[0]:=Sensor_Reading_2[3];
TemperatureSensors_2:=DINT_TO_LREAL(LREAL_TO_DINT(dut_sensor_datas_2.data_lreal*100))/100;
//sensor_3
dut_sensor_datas_3.data_byte[3]:=Sensor_Reading_3[0];
dut_sensor_datas_3.data_byte[2]:=Sensor_Reading_3[1];
dut_sensor_datas_3.data_byte[1]:=Sensor_Reading_3[2];
dut_sensor_datas_3.data_byte[0]:=Sensor_Reading_3[3];
TemperatureSensors_3:=DINT_TO_LREAL(LREAL_TO_DINT(dut_sensor_datas_3.data_lreal*100))/100;
//sensor_4
dut_sensor_datas_4.data_byte[3]:=Sensor_Reading_4[0];
dut_sensor_datas_4.data_byte[2]:=Sensor_Reading_4[1];
dut_sensor_datas_4.data_byte[1]:=Sensor_Reading_4[2];
dut_sensor_datas_4.data_byte[0]:=Sensor_Reading_4[3];
TemperatureSensors_4:=DINT_TO_LREAL(LREAL_TO_DINT(dut_sensor_datas_4.data_lreal*100))/100;
//sensor_5
dut_sensor_datas_5.data_byte[3]:=Sensor_Reading_5[0];
dut_sensor_datas_5.data_byte[2]:=Sensor_Reading_5[1];
dut_sensor_datas_5.data_byte[1]:=Sensor_Reading_5[2];
dut_sensor_datas_5.data_byte[0]:=Sensor_Reading_5[3];
TemperatureSensors_5:=DINT_TO_LREAL(LREAL_TO_DINT(dut_sensor_datas_5.data_lreal*100))/100;
//sensor_6
dut_sensor_datas_6.data_byte[3]:=Sensor_Reading_6[0];
dut_sensor_datas_6.data_byte[2]:=Sensor_Reading_6[1];
dut_sensor_datas_6.data_byte[1]:=Sensor_Reading_6[2];
dut_sensor_datas_6.data_byte[0]:=Sensor_Reading_6[3];
TemperatureSensors_6:=DINT_TO_LREAL(LREAL_TO_DINT(dut_sensor_datas_6.data_lreal*100))/100;
//sensor_7
dut_sensor_datas_7.data_byte[3]:=Sensor_Reading_7[0];
dut_sensor_datas_7.data_byte[2]:=Sensor_Reading_7[1];
dut_sensor_datas_7.data_byte[1]:=Sensor_Reading_7[2];
dut_sensor_datas_7.data_byte[0]:=Sensor_Reading_7[3];
TemperatureSensors_7:=DINT_TO_LREAL(LREAL_TO_DINT(dut_sensor_datas_7.data_lreal*100))/100;
//sensor_8
dut_sensor_datas_8.data_byte[3]:=Sensor_Reading_8[0];
dut_sensor_datas_8.data_byte[2]:=Sensor_Reading_8[1];
dut_sensor_datas_8.data_byte[1]:=Sensor_Reading_8[2];
dut_sensor_datas_8.data_byte[0]:=Sensor_Reading_8[3];
TemperatureSensors_8:=DINT_TO_LREAL(LREAL_TO_DINT(dut_sensor_datas_8.data_lreal*100))/100;
//计算temperature_gradient
temperature_gradient_2_To_1:=ABS(TemperatureSensors_2-TemperatureSensors_1);
temperature_gradient_3_To_2:=ABS(TemperatureSensors_3-TemperatureSensors_2);
temperature_gradient_5_To_4:=ABS(TemperatureSensors_5-TemperatureSensors_4);
temperature_gradient_6_To_5:=ABS(TemperatureSensors_6-TemperatureSensors_5);
temperature_gradient_max:=DINT_TO_LREAL(LREAL_TO_DINT(MAX(temperature_gradient_2_To_1,temperature_gradient_3_To_2,
							temperature_gradient_5_To_4,temperature_gradient_6_To_5)*100))/100;
//计算大梁上的温度平均值
temperature_average:=DINT_TO_LREAL(LREAL_TO_DINT((TemperatureSensors_1+TemperatureSensors_2+TemperatureSensors_3+TemperatureSensors_4
					+TemperatureSensors_5+TemperatureSensors_6)/6*100))/100;
					

//传感器温度状态：0：有传感器度数错误；1:常温；2:低温；3:常温和低温中间态
IF TemperatureSensors_1=0 OR TemperatureSensors_2=0 OR TemperatureSensors_3=0 
	OR TemperatureSensors_4=0 OR TemperatureSensors_5=0 OR TemperatureSensors_6=0 THEN	
	temperatureStatus:=0;//有传感器读数错误
ELSIF TemperatureSensors_1>=RoomTemperatureThreshold AND TemperatureSensors_2>=RoomTemperatureThreshold AND TemperatureSensors_3>=RoomTemperatureThreshold
	AND TemperatureSensors_4>=RoomTemperatureThreshold AND TemperatureSensors_5>=RoomTemperatureThreshold AND TemperatureSensors_6>=RoomTemperatureThreshold THEN	
	temperatureStatus:=1;//常温
ELSIF TemperatureSensors_1<=CryogenicTemperatureThreshold AND TemperatureSensors_1>77
	AND TemperatureSensors_2<=CryogenicTemperatureThreshold  AND TemperatureSensors_2>77
	AND TemperatureSensors_3<=CryogenicTemperatureThreshold  AND TemperatureSensors_3>77
	AND TemperatureSensors_4<=CryogenicTemperatureThreshold   AND TemperatureSensors_4>77
	AND TemperatureSensors_5<=CryogenicTemperatureThreshold  AND TemperatureSensors_5>77
	AND TemperatureSensors_6<=CryogenicTemperatureThreshold   AND TemperatureSensors_6>77 THEN	
	temperatureStatus:=2;//低温
ELSE
	temperatureStatus:=3;//常温和低温中间
END_IF
END_ACTION

ACTION A_InitAxisParameters:
//LE
	Pos_LeftTopLin:=DINT_TO_LREAL(LREAL_TO_DINT(LeftTopLin.NcToPlc.ActPos*100000))/100000;
	Pos_RightTopLin:=DINT_TO_LREAL(LREAL_TO_DINT(RightTopLin.NcToPlc.ActPos*100000))/100000;
	Pos_LeftBottomLin:=DINT_TO_LREAL(LREAL_TO_DINT(LeftBottomLin.NcToPlc.ActPos*100000))/100000;
	Pos_RightBottomLin:=DINT_TO_LREAL(LREAL_TO_DINT(RightBottomLin.NcToPlc.ActPos*100000))/100000;	
	Pos_LeftInLin:=DINT_TO_LREAL(LREAL_TO_DINT(LeftInLin.NcToPlc.ActPos*100000))/100000;
	Pos_RightInLin:=DINT_TO_LREAL(LREAL_TO_DINT(RightInLin.NcToPlc.ActPos*100000))/100000;
	Pos_LeftOutLin:=DINT_TO_LREAL(LREAL_TO_DINT(LeftOutLin.NcToPlc.ActPos*100000))/100000;
	Pos_RightOutLin:=DINT_TO_LREAL(LREAL_TO_DINT(RightOutLin.NcToPlc.ActPos*100000))/100000;

	moveStatusLeftTop:=LeftTopLin.Status.Moving;
	moveStatusRightTop:=RightTopLin.Status.Moving;
	moveStatusLeftBottom:=LeftBottomLin.Status.Moving;
	moveStatusRightBottom:=RightBottomLin.Status.Moving;
	moveStatusLeftIn:=LeftInLin.Status.Moving;
	moveStatusRightIn:=RightInLin.Status.Moving;
	moveStatusLeftOut:=LeftOutLin.Status.Moving;
	moveStatusRightOut:=RightOutLin.Status.Moving;
	moveStatusAllAxis:=moveStatusLeftTop AND moveStatusRightTop AND moveStatusLeftBottom AND moveStatusRightBottom
						AND moveStatusLeftIn AND moveStatusRightIn AND moveStatusLeftOut AND moveStatusRightOut;
	moveStatusAnyAxis:=moveStatusLeftTop OR moveStatusRightTop OR moveStatusLeftBottom OR moveStatusRightBottom
						OR moveStatusLeftIn OR moveStatusRightIn OR moveStatusLeftOut OR moveStatusRightOut;
						
	Velo_LeftTopLin:=DINT_TO_LREAL(LREAL_TO_DINT(LeftTopLin.NcToPlc.ActVelo*100000))/100000;
	Velo_RightTopLin:=DINT_TO_LREAL(LREAL_TO_DINT(RightTopLin.NcToPlc.ActVelo*100000))/100000;
	Velo_LeftBottomLin:=DINT_TO_LREAL(LREAL_TO_DINT(LeftBottomLin.NcToPlc.ActVelo*100000))/100000;
	Velo_RightBottomLin:=DINT_TO_LREAL(LREAL_TO_DINT(RightBottomLin.NcToPlc.ActVelo*100000))/100000;
	Velo_LeftInLin:=DINT_TO_LREAL(LREAL_TO_DINT(LeftInLin.NcToPlc.ActVelo*100000))/100000;
	Velo_RightInLin:=DINT_TO_LREAL(LREAL_TO_DINT(RightInLin.NcToPlc.ActVelo*100000))/100000;
	Velo_LeftOutLin:=DINT_TO_LREAL(LREAL_TO_DINT(LeftOutLin.NcToPlc.ActVelo*100000))/100000;
	Velo_RightOutLin:=DINT_TO_LREAL(LREAL_TO_DINT(RightOutLin.NcToPlc.ActVelo*100000))/100000;

	PosDiff_LeftTopLin_actual:=DINT_TO_LREAL(LREAL_TO_DINT(LeftTopLin.NcToPlc.PosDiff*100000))/100000;
	PosDiff_RightTopLin_actual:=DINT_TO_LREAL(LREAL_TO_DINT(RightTopLin.NcToPlc.PosDiff*100000))/100000;
	PosDiff_LeftBottomLin_actual:=DINT_TO_LREAL(LREAL_TO_DINT(LeftBottomLin.NcToPlc.PosDiff*100000))/100000;
	PosDiff_RightBottomLin_actual:=DINT_TO_LREAL(LREAL_TO_DINT(RightBottomLin.NcToPlc.PosDiff*100000))/100000;
	PosDiff_LeftInLin_actual:=DINT_TO_LREAL(LREAL_TO_DINT(LeftInLin.NcToPlc.PosDiff*100000))/100000;
	PosDiff_RightInLin_actual:=DINT_TO_LREAL(LREAL_TO_DINT(RightInLin.NcToPlc.PosDiff*100000))/100000;
	PosDiff_LeftOutLin_actual:=DINT_TO_LREAL(LREAL_TO_DINT(LeftOutLin.NcToPlc.PosDiff*100000))/100000;
	PosDiff_RightOutLin_actual:=DINT_TO_LREAL(LREAL_TO_DINT(RightOutLin.NcToPlc.PosDiff*100000))/100000;

	Torque_LeftTopLin:=DINT_TO_LREAL(LREAL_TO_DINT(LeftTopLin.NcToPlc.ActTorque*100000))/100000;
	Torque_RightTopLin:=DINT_TO_LREAL(LREAL_TO_DINT(RightTopLin.NcToPlc.ActTorque*100000))/100000;
	Torque_LeftBottomLin:=DINT_TO_LREAL(LREAL_TO_DINT(LeftBottomLin.NcToPlc.ActTorque*100000))/100000;
	Torque_RightBottomLin:=DINT_TO_LREAL(LREAL_TO_DINT(RightBottomLin.NcToPlc.ActTorque*100000))/100000;
	Torque_LeftInLin:=DINT_TO_LREAL(LREAL_TO_DINT(LeftInLin.NcToPlc.ActTorque*100000))/100000;
	Torque_RightInLin:=DINT_TO_LREAL(LREAL_TO_DINT(RightInLin.NcToPlc.ActTorque*100000))/100000;
	Torque_LeftOutLin:=DINT_TO_LREAL(LREAL_TO_DINT(LeftOutLin.NcToPlc.ActTorque*100000))/100000;
	Torque_RightOutLin:=DINT_TO_LREAL(LREAL_TO_DINT(RightOutLin.NcToPlc.ActTorque*100000))/100000;
	
	LeftTopLin.ReadStatus();
	RightTopLin.ReadStatus();
	LeftBottomLin.ReadStatus();
	RightBottomLin.ReadStatus();
	LeftInLin.ReadStatus();
	RightInLin.ReadStatus();
	LeftOutLin.ReadStatus();
	RightOutLin.ReadStatus();

	//Motor

	Pos_LeftTopMotor:=DINT_TO_LREAL(LREAL_TO_DINT(LeftTopMotor.NcToPlc.ActPos*100000))/100000;
	Pos_RightTopMotor:=DINT_TO_LREAL(LREAL_TO_DINT(RightTopMotor.NcToPlc.ActPos*100000))/100000;
	Pos_LeftBottomMotor:=DINT_TO_LREAL(LREAL_TO_DINT(LeftBottomMotor.NcToPlc.ActPos*100000))/100000;
	Pos_RightBottomMotor:=DINT_TO_LREAL(LREAL_TO_DINT(RightBottomMotor.NcToPlc.ActPos*100000))/100000;	
	Pos_LeftInMotor:=DINT_TO_LREAL(LREAL_TO_DINT(LeftInMotor.NcToPlc.ActPos*100000))/100000;
	Pos_RightInMotor:=DINT_TO_LREAL(LREAL_TO_DINT(RightInMotor.NcToPlc.ActPos*100000))/100000;
	Pos_LeftOutMotor:=DINT_TO_LREAL(LREAL_TO_DINT(LeftOutMotor.NcToPlc.ActPos*100000))/100000;
	Pos_RightOutMotor:=DINT_TO_LREAL(LREAL_TO_DINT(RightOutMotor.NcToPlc.ActPos*100000))/100000;

	moveStatusLeftTop:=LeftTopMotor.Status.Moving;
	moveStatusRightTop:=RightTopMotor.Status.Moving;
	moveStatusLeftBottom:=LeftBottomMotor.Status.Moving;
	moveStatusRightBottom:=RightBottomMotor.Status.Moving;
	moveStatusLeftIn:=LeftInMotor.Status.Moving;
	moveStatusRightIn:=RightInMotor.Status.Moving;
	moveStatusLeftOut:=LeftOutMotor.Status.Moving;
	moveStatusRightOut:=RightOutMotor.Status.Moving;
	moveStatusAllAxis:=moveStatusLeftTop AND moveStatusRightTop AND moveStatusLeftBottom AND moveStatusRightBottom
						AND moveStatusLeftIn AND moveStatusRightIn AND moveStatusLeftOut AND moveStatusRightOut;
	moveStatusAnyAxis:=moveStatusLeftTop OR moveStatusRightTop OR moveStatusLeftBottom OR moveStatusRightBottom
						OR moveStatusLeftIn OR moveStatusRightIn OR moveStatusLeftOut OR moveStatusRightOut;
						
	Velo_LeftTopMotor:=DINT_TO_LREAL(LREAL_TO_DINT(LeftTopMotor.NcToPlc.ActVelo*100000))/100000;
	Velo_RightTopMotor:=DINT_TO_LREAL(LREAL_TO_DINT(RightTopMotor.NcToPlc.ActVelo*100000))/100000;
	Velo_LeftBottomMotor:=DINT_TO_LREAL(LREAL_TO_DINT(LeftBottomMotor.NcToPlc.ActVelo*100000))/100000;
	Velo_RightBottomMotor:=DINT_TO_LREAL(LREAL_TO_DINT(RightBottomMotor.NcToPlc.ActVelo*100000))/100000;
	Velo_LeftInMotor:=DINT_TO_LREAL(LREAL_TO_DINT(LeftInMotor.NcToPlc.ActVelo*100000))/100000;
	Velo_RightInMotor:=DINT_TO_LREAL(LREAL_TO_DINT(RightInMotor.NcToPlc.ActVelo*100000))/100000;
	Velo_LeftOutMotor:=DINT_TO_LREAL(LREAL_TO_DINT(LeftOutMotor.NcToPlc.ActVelo*100000))/100000;
	Velo_RightOutMotor:=DINT_TO_LREAL(LREAL_TO_DINT(RightOutMotor.NcToPlc.ActVelo*100000))/100000;

	PosDiff_LeftTopMotor_actual:=DINT_TO_LREAL(LREAL_TO_DINT(LeftTopMotor.NcToPlc.PosDiff*100000))/100000;
	PosDiff_RightTopMotor_actual:=DINT_TO_LREAL(LREAL_TO_DINT(RightTopMotor.NcToPlc.PosDiff*100000))/100000;
	PosDiff_LeftBottomMotor_actual:=DINT_TO_LREAL(LREAL_TO_DINT(LeftBottomMotor.NcToPlc.PosDiff*100000))/100000;
	PosDiff_RightBottomMotor_actual:=DINT_TO_LREAL(LREAL_TO_DINT(RightBottomMotor.NcToPlc.PosDiff*100000))/100000;
	PosDiff_LeftInMotor_actual:=DINT_TO_LREAL(LREAL_TO_DINT(LeftInMotor.NcToPlc.PosDiff*100000))/100000;
	PosDiff_RightInMotor_actual:=DINT_TO_LREAL(LREAL_TO_DINT(RightInMotor.NcToPlc.PosDiff*100000))/100000;
	PosDiff_LeftOutMotor_actual:=DINT_TO_LREAL(LREAL_TO_DINT(LeftOutMotor.NcToPlc.PosDiff*100000))/100000;
	PosDiff_RightOutMotor_actual:=DINT_TO_LREAL(LREAL_TO_DINT(RightOutMotor.NcToPlc.PosDiff*100000))/100000;

	Torque_LeftTopMotor:=DINT_TO_LREAL(LREAL_TO_DINT(LeftTopMotor.NcToPlc.ActTorque*100000))/100000;
	Torque_RightTopMotor:=DINT_TO_LREAL(LREAL_TO_DINT(RightTopMotor.NcToPlc.ActTorque*100000))/100000;
	Torque_LeftBottomMotor:=DINT_TO_LREAL(LREAL_TO_DINT(LeftBottomMotor.NcToPlc.ActTorque*100000))/100000;
	Torque_RightBottomMotor:=DINT_TO_LREAL(LREAL_TO_DINT(RightBottomMotor.NcToPlc.ActTorque*100000))/100000;
	Torque_LeftInMotor:=DINT_TO_LREAL(LREAL_TO_DINT(LeftInMotor.NcToPlc.ActTorque*100000))/100000;
	Torque_RightInMotor:=DINT_TO_LREAL(LREAL_TO_DINT(RightInMotor.NcToPlc.ActTorque*100000))/100000;
	Torque_LeftOutMotor:=DINT_TO_LREAL(LREAL_TO_DINT(LeftOutMotor.NcToPlc.ActTorque*100000))/100000;
	Torque_RightOutMotor:=DINT_TO_LREAL(LREAL_TO_DINT(RightOutMotor.NcToPlc.ActTorque*100000))/100000;
	
	LeftTopMotor.ReadStatus();
	RightTopMotor.ReadStatus();
	LeftBottomMotor.ReadStatus();
	RightBottomMotor.ReadStatus();
	LeftInMotor.ReadStatus();
	RightInMotor.ReadStatus();
	LeftOutMotor.ReadStatus();
	RightOutMotor.ReadStatus();
	//
	//get Delta
	//
	//Delta Pos
	DeltaPos_LeftTop:=Pos_LeftTopLin - Pos_LeftTopMotor;
	DeltaPos_RightTop:=Pos_RightTopLin - Pos_RightTopMotor;
	DeltaPos_LeftBottom:=Pos_LeftBottomLin - Pos_LeftBottomMotor;
	DeltaPos_RightBottom:=Pos_RightBottomLin - Pos_RightBottomMotor;
	DeltaPos_LeftIn:=Pos_LeftInLin - Pos_LeftInMotor;
	DeltaPos_RightIn:=Pos_RightInLin - Pos_RightInMotor;
	DeltaPos_LeftOut:=Pos_LeftOutLin - Pos_LeftOutMotor;
	DeltaPos_RightOut:=Pos_RightOutLin - Pos_RightOutMotor;
	//Delta Velocity	
	DeltaVelo_LeftTop:=Velo_LeftTopLin - Velo_LeftTopMotor;
	DeltaVelo_RightTop:=Velo_RightTopLin - Velo_RightTopMotor;
	DeltaVelo_LeftBottom:=Velo_LeftBottomLin - Velo_LeftBottomMotor;
	DeltaVelo_RightBottom:=Velo_RightBottomLin - Velo_RightBottomMotor;	
	DeltaVelo_LeftIn:=Velo_LeftInLin - Velo_LeftInMotor;
	DeltaVelo_RightIn:=Velo_RightInLin - Velo_RightInMotor;
	DeltaVelo_LeftOut:=Velo_LeftOutLin - Velo_LeftOutMotor;
	DeltaVelo_RightOut:=Velo_RightOutLin - Velo_RightOutMotor;
	//Delta lagDistance
	DeltaPosDiff_LeftTop_actual:=PosDiff_LeftTopLin_actual - PosDiff_LeftTopMotor_actual;
	DeltaPosDiff_RightTop_actual:=PosDiff_RightTopLin_actual - PosDiff_RightTopMotor_actual;
	DeltaPosDiff_LeftBottom_actual:=PosDiff_LeftBottomLin_actual - PosDiff_LeftBottomMotor_actual;
	DeltaPosDiff_RightBottom_actual:=PosDiff_RightBottomLin_actual - PosDiff_RightBottomMotor_actual;	
	DeltaPosDiff_LeftIn_actual:=PosDiff_LeftInLin_actual - PosDiff_LeftInMotor_actual;
	DeltaPosDiff_RightIn_actual:=PosDiff_RightInLin_actual - PosDiff_RightInMotor_actual;
	DeltaPosDiff_LeftOut_actual:=PosDiff_LeftOutLin_actual - PosDiff_LeftOutMotor_actual;
	DeltaPosDiff_RightOut_actual:=PosDiff_RightOutLin_actual - PosDiff_RightOutMotor_actual;
	//Delta Torque
	DeltaTorque_LeftTop:=Torque_LeftTopLin - Torque_LeftTopMotor;
	DeltaTorque_RightTop:=Torque_RightTopLin - Torque_RightTopMotor;
	DeltaTorque_LeftBottom:=Torque_LeftBottomLin -Torque_LeftBottomMotor;
	DeltaTorque_RightBottom:=Torque_RightBottomLin - Torque_RightBottomMotor;
	DeltaTorque_LeftIn:=Torque_LeftInLin - Torque_LeftInMotor;
	DeltaTorque_RightIn:=Torque_RightInLin - Torque_RightInMotor;
	DeltaTorque_LeftOut:=Torque_LeftOutLin -Torque_LeftOutMotor;
	DeltaTorque_RightOut:=Torque_RightOutLin - Torque_RightOutMotor;
END_ACTION

ACTION A_InitRecipeParameters:
CASE state_loadParameters OF
	0:
		LoadParameter:=TRUE;
		Read_R_TRIG(CLK:=LoadParameter , Q=> );
		IF Read_R_TRIG.Q THEN
			state_loadParameters:=1;
		END_IF
	1:
		 ReturnDwordLoad:=RecipeManCommands.LoadAndWriteRecipe(RecipeDefinitionName:='Recipes' , RecipeName:='ParametersIAMW');
    	 LoadParameter:=FALSE;
		 IF ReturnDwordLoad<>0 THEN
		 	state_loadParameters:=-100;
		ELSE
			LoadRecipeParameters:=TRUE;
			LoadParameter:=FALSE;
			state_loadParameters:=88;
	 	END_IF
	88:
		loadParametersDone:=TRUE;
	-100:
		loadParametersDone:=FALSE;
		Error:=TRUE;
		ErrorId:=101;
		ErrorDescription:='LoadRecipeParameters Error';
		Plc_EmergencyStop:=FALSE;
END_CASE
(*
Save_R_TRIG(CLK:=SaveParameter , Q=> );
Read_R_TRIG(CLK:=LoadParameter , Q=> );
IF Save_R_TRIG.Q THEN  //将plc数据以文件形式保存在工控机中
	 RecipeManCommands.CreateRecipe(RecipeDefinitionName:='Recipes' , RecipeName:='ParametersIAMW' );
	 RecipeManCommands.ReadAndSaveRecipe(RecipeDefinitionName:='Recipes' , RecipeName:='ParametersIAMW' );
	 SaveParameter:=FALSE;
END_IF
//IF Read_R_TRIG.Q THEN  //将工控机中的文件数据读取到plc中
//     ReturnDwordLoad:=RecipeManCommands.LoadAndWriteRecipe(RecipeDefinitionName:='Recipes' , RecipeName:='Parameters');
//     LoadParameter:=FALSE;
//	 IF ReturnDwordLoad<>0 THEN
//		 Error:=TRUE;
//		 ErrorId:=101;
//		 ErrorDescription:='LoadRecipeParameters Error';
//		 Plc_EmergencyStop:=FALSE;
//	 END_IF
//END_IF 
*)
END_ACTION

ACTION A_KillOpcIocShellExe:
R_TRIG_Exekill(CLK:=bExe_Kill_Prog, Q=> );
CASE Exe_kill_step OF
	0:
		IF R_TRIG_Exekill.Q THEN
			NT_StartProcess_Kill.START:=FALSE;
			NT_StartProcess_Kill.PATHSTR:='C:\HZB\OpcIocShell\IDControlIOC\killcmd.bat';
			//NT_StartProcess_Kill.DIRNAME:='C:\Program Files (x86)\HZB\OpcIocShell\bin\opcIocShell.exe';
			Exe_kill_step:=10;
		END_IF;
	10:
		NT_StartProcess_Kill.START:=TRUE;
		Exe_kill_step:=20;
	20:
		IF NT_StartProcess_Kill.ERR THEN
			Exe_kill_step:=0;
		ELSE
			Exe_kill_step:=30;
		END_IF;

	30:
		NT_StartProcess_Kill.START:=TRUE;
		Exe_kill_step:=40;
	40:
		IF NOT NT_StartProcess_Kill.BUSY THEN
			NT_StartProcess_Kill.START:=FALSE;
			Exe_Kill_Done:=TRUE;
			Exe_kill_step:=0;
		END_IF;
END_CASE;

NT_StartProcess_Kill(
	NETID:='' ,
	PATHSTR:= ,
	DIRNAME:= , 
	COMNDLINE:= , 
	START:= ,
	ERRID=> );
END_ACTION

ACTION A_LEHeartBeatMonitor:
//monitor only while power on and not simulation or not use LE
IF NOT st_Power THEN
	RETURN;
END_IF
(**)
IF simulation THEN
	RETURN;
END_IF
IF NOT USELinearEncoder THEN
	RETURN;
END_IF

// 初始化
IF LEHeartBeatFirstScan THEN
    Velo_LeftTopLin_Last := LeftTopLin.NcToPlc.ActVelo;
    Velo_RightTopLin_Last := RightTopLin.NcToPlc.ActVelo;
    Velo_LeftBottomLin_Last := LeftBottomLin.NcToPlc.ActVelo;
    Velo_RightBottomLin_Last := RightBottomLin.NcToPlc.ActVelo;
    Velo_LeftInLin_Last := LeftInLin.NcToPlc.ActVelo;
    Velo_RightInLin_Last := RightInLin.NcToPlc.ActVelo;
    Velo_LeftOutLin_Last := LeftOutLin.NcToPlc.ActVelo;
    Velo_RightOutLin_Last := RightOutLin.NcToPlc.ActVelo;
    LEHeartBeatFirstScan := FALSE;
END_IF;

// 计算光栅前后速度差，速度差比位置差更敏感
DeltaVelo_LeftTopLin := ABS(LeftTopLin.NcToPlc.ActVelo - Velo_LeftTopLin_Last);
DeltaVelo_RightTopLin := ABS(RightTopLin.NcToPlc.ActVelo - Velo_RightTopLin_Last);
DeltaVelo_LeftBottomLin := ABS(LeftBottomLin.NcToPlc.ActVelo - Velo_LeftBottomLin_Last);
DeltaVelo_RightBottomLin := ABS(RightBottomLin.NcToPlc.ActVelo - Velo_RightBottomLin_Last);
DeltaVelo_LeftInLin := ABS(LeftInLin.NcToPlc.ActVelo - Velo_LeftInLin_Last);
DeltaVelo_RightInLin := ABS(RightInLin.NcToPlc.ActVelo - Velo_RightInLin_Last);
DeltaVelo_LeftOutLin := ABS(LeftOutLin.NcToPlc.ActVelo - Velo_LeftOutLin_Last);
DeltaVelo_RightOutLin := ABS(RightOutLin.NcToPlc.ActVelo - Velo_RightOutLin_Last);
//LeftTop monitor
IF DeltaVelo_LeftTopLin > LEHeartBeatDeadZone THEN
    // 有变动，光栅正常，计数器归零，更新位置,重置所有状态
    StableTimer_LeftTopLin(IN := FALSE, PT := LEHeartBeatAlarmTime);
    Alarm_LeftTopLin := FALSE;
    Velo_LeftTopLin_Last := LeftTopLin.NcToPlc.ActVelo;  // 
    StableTime_LeftTopLin := T#0S;
	IsInitialPositionSet_LeftTop:=FALSE;
	Alarm_LeftTopMotorPos:=FALSE;
	Alarm_LeftTopMotorVelo:=FALSE;
ELSE
    //一点变动没有了，光栅异常，开始计时
    StableTimer_LeftTopLin(
        IN := TRUE,
        PT := LEHeartBeatAlarmTime,
        ET => StableTime_LeftTopLin
    );
	//记录电机初始位置，后后续对比做准备
	IF NOT IsInitialPositionSet_LeftTop THEN
        Pos_LeftTopMotor_Initial := Pos_LeftTopMotor;  // 记录初始位置
        IsInitialPositionSet_LeftTop := TRUE;
   	END_IF;
    
    // 100ms速度完全不变，开始监控电机速度和位置
    IF StableTimer_LeftTopLin.Q THEN
        Alarm_LeftTopLin := TRUE;  // 
			//电机位置对比及监测
			MotorPosChange_LeftTop:=ABS( Pos_LeftTopMotor-Pos_LeftTopMotor_Initial);
			IF MotorPosChange_LeftTop > Threshold_LeftTopMotorPos THEN
				Alarm_LeftTopMotorPos:=TRUE;
				ErrorID:=5001;
				ErrorDescription:='5001';
				Error:=TRUE;
				FB_PlcEmergencyStop();
				LED_Error:=TRUE;
			ELSE
				Alarm_LeftTopMotorPos:=FALSE;
			END_IF
			//电机速度监测
			IF Velo_LeftTopMotor > Threshold_LeftTopMotorVelo THEN
				Alarm_LeftTopMotorVelo:=TRUE;
				ErrorID:=5002;
				ErrorDescription:='5002';
				Error:=TRUE;
				FB_PlcEmergencyStop();
				LED_Error:=TRUE;
			ELSE
				Alarm_LeftTopMotorVelo:=FALSE;
			END_IF
    ELSE
        Alarm_LeftTopLin := FALSE;
	END_IF
END_IF
//RightTop monitor
IF DeltaVelo_RightTopLin > LEHeartBeatDeadZone THEN
    // 有变动，光栅正常，计数器归零，更新位置,重置所有状态
    StableTimer_RightTopLin(IN := FALSE, PT := LEHeartBeatAlarmTime);
    Alarm_RightTopLin := FALSE;
    Velo_RightTopLin_Last := RightTopLin.NcToPlc.ActVelo;  // 
    StableTime_RightTopLin := T#0S;
	IsInitialPositionSet_RightTop:=FALSE;
	Alarm_RightTopMotorPos:=FALSE;
	Alarm_RightTopMotorVelo:=FALSE;
ELSE
    //一点变动没有了，光栅异常，开始计时
    StableTimer_RightTopLin(
        IN := TRUE,
        PT :=LEHeartBeatAlarmTime,
        ET => StableTime_RightTopLin
    );
	//记录电机初始位置，后后续对比做准备
	IF NOT IsInitialPositionSet_RightTop THEN
        Pos_RightTopMotor_Initial := Pos_RightTopMotor;  // 记录初始位置
        IsInitialPositionSet_RightTop := TRUE;
   	END_IF;
    
    // 100ms速度完全不变，开始监控电机速度和位置
    IF StableTimer_RightTopLin.Q THEN
        Alarm_RightTopLin := TRUE;  // 
			//电机位置对比及监测
			MotorPosChange_RightTop:=ABS( Pos_RightTopMotor-Pos_RightTopMotor_Initial);
			IF MotorPosChange_RightTop > Threshold_RightTopMotorPos THEN
				Alarm_RightTopMotorPos:=TRUE;
				ErrorID:=5003;
				ErrorDescription:='5003';
				Error:=TRUE;
				FB_PlcEmergencyStop();
				LED_Error:=TRUE;
			ELSE
				Alarm_RightTopMotorPos:=FALSE;
			END_IF
			//电机速度监测
			IF Velo_RightTopMotor > Threshold_RightTopMotorVelo THEN
				Alarm_RightTopMotorVelo:=TRUE;
				ErrorID:=5004;
				ErrorDescription:='5004';
				Error:=TRUE;
				FB_PlcEmergencyStop();
				LED_Error:=TRUE;
			ELSE
				Alarm_RightTopMotorVelo:=FALSE;
			END_IF
    ELSE
        Alarm_RightTopLin := FALSE;
	END_IF
END_IF
//LeftBottom monitor
IF DeltaVelo_LeftBottomLin > LEHeartBeatDeadZone THEN
    // 有变动，光栅正常，计数器归零，更新位置,重置所有状态
    StableTimer_LeftBottomLin(IN := FALSE, PT := LEHeartBeatAlarmTime);
    Alarm_LeftBottomLin := FALSE;
    Velo_LeftBottomLin_Last := LeftBottomLin.NcToPlc.ActVelo;  // 
    StableTime_LeftBottomLin := T#0S;
	IsInitialPositionSet_LeftBottom:=FALSE;
	Alarm_LeftBottomMotorPos:=FALSE;
	Alarm_LeftBottomMotorVelo:=FALSE;
ELSE
    //一点变动没有了，光栅异常，开始计时
    StableTimer_LeftBottomLin(
        IN := TRUE,
        PT := LEHeartBeatAlarmTime,
        ET => StableTime_LeftBottomLin
    );
	//记录电机初始位置，后后续对比做准备
	IF NOT IsInitialPositionSet_LeftBottom THEN
        Pos_LeftBottomMotor_Initial := Pos_LeftBottomMotor;  // 记录初始位置
        IsInitialPositionSet_LeftBottom := TRUE;
   	END_IF;
    
    // 100ms速度完全不变，开始监控电机速度和位置
    IF StableTimer_LeftBottomLin.Q THEN
        Alarm_LeftBottomLin := TRUE;  // 
			//电机位置对比及监测
			MotorPosChange_LeftBottom:=ABS( Pos_LeftBottomMotor-Pos_LeftBottomMotor_Initial);
			IF MotorPosChange_LeftBottom > Threshold_LeftBottomMotorPos THEN
				Alarm_LeftBottomMotorPos:=TRUE;
				ErrorID:=5005;
				ErrorDescription:='5005';
				Error:=TRUE;
				FB_PlcEmergencyStop();
				LED_Error:=TRUE;
			ELSE
				Alarm_LeftBottomMotorPos:=FALSE;
			END_IF
			//电机速度监测
			IF Velo_LeftBottomMotor > Threshold_LeftBottomMotorVelo THEN
				Alarm_LeftBottomMotorVelo:=TRUE;
				ErrorID:=5006;
				ErrorDescription:='5006';
				Error:=TRUE;
				FB_PlcEmergencyStop();
				LED_Error:=TRUE;
			ELSE
				Alarm_LeftBottomMotorVelo:=FALSE;
			END_IF
    ELSE
        Alarm_LeftBottomLin := FALSE;
	END_IF
END_IF
//RightBottom monitor
IF DeltaVelo_RightBottomLin > LEHeartBeatDeadZone THEN
    // 有变动，光栅正常，计数器归零，更新位置,重置所有状态
    StableTimer_RightBottomLin(IN := FALSE, PT := LEHeartBeatAlarmTime);
    Alarm_RightBottomLin := FALSE;
    Velo_RightBottomLin_Last := RightBottomLin.NcToPlc.ActVelo;  // 
    StableTime_RightBottomLin := T#0S;
	IsInitialPositionSet_RightBottom:=FALSE;
	Alarm_RightBottomMotorPos:=FALSE;
	Alarm_RightBottomMotorVelo:=FALSE;
ELSE
    //一点变动没有了，光栅异常，开始计时
    StableTimer_RightBottomLin(
        IN := TRUE,
        PT := LEHeartBeatAlarmTime,
        ET => StableTime_RightBottomLin
    );
	//记录电机初始位置，后后续对比做准备
	IF NOT IsInitialPositionSet_RightBottom THEN
        Pos_RightBottomMotor_Initial := Pos_RightBottomMotor;  // 记录初始位置
        IsInitialPositionSet_RightBottom := TRUE;
   	END_IF;
    
    // 100ms速度完全不变，开始监控电机速度和位置
    IF StableTimer_RightBottomLin.Q THEN
        Alarm_RightBottomLin := TRUE;  // 
			//电机位置对比及监测
			MotorPosChange_RightBottom:=ABS( Pos_RightBottomMotor-Pos_RightBottomMotor_Initial);
			IF MotorPosChange_RightBottom > Threshold_RightBottomMotorPos THEN
				Alarm_RightBottomMotorPos:=TRUE;
				ErrorID:=5007;
				ErrorDescription:='5007';
				Error:=TRUE;
				FB_PlcEmergencyStop();
				LED_Error:=TRUE;
			ELSE
				Alarm_RightBottomMotorPos:=FALSE;
			END_IF
			//电机速度监测
			IF Velo_RightBottomMotor > Threshold_RightBottomMotorVelo THEN
				Alarm_RightBottomMotorVelo:=TRUE;
				ErrorID:=5008;
				ErrorDescription:='5008';
				Error:=TRUE;
				FB_PlcEmergencyStop();
				LED_Error:=TRUE;
			ELSE
				Alarm_RightBottomMotorVelo:=FALSE;
			END_IF
    ELSE
        Alarm_RightBottomLin := FALSE;
	END_IF
END_IF
//LeftIn monitor
IF DeltaVelo_LeftInLin > LEHeartBeatDeadZone THEN
    // 有变动，光栅正常，计数器归零，更新位置,重置所有状态
    StableTimer_LeftInLin(IN := FALSE, PT := LEHeartBeatAlarmTime);
    Alarm_LeftInLin := FALSE;
    Velo_LeftInLin_Last := LeftInLin.NcToPlc.ActVelo;  // 
    StableTime_LeftInLin := T#0S;
	IsInitialPositionSet_LeftIn:=FALSE;
	Alarm_LeftInMotorPos:=FALSE;
	Alarm_LeftInMotorVelo:=FALSE;
ELSE
    //一点变动没有了，光栅异常，开始计时
    StableTimer_LeftInLin(
        IN := TRUE,
        PT := LEHeartBeatAlarmTime,
        ET => StableTime_LeftInLin
    );
	//记录电机初始位置，后后续对比做准备
	IF NOT IsInitialPositionSet_LeftIn THEN
        Pos_LeftInMotor_Initial := Pos_LeftInMotor;  // 记录初始位置
        IsInitialPositionSet_LeftIn := TRUE;
   	END_IF;
    
    // 100ms速度完全不变，开始监控电机速度和位置
    IF StableTimer_LeftInLin.Q THEN
        Alarm_LeftInLin := TRUE;  // 
			//电机位置对比及监测
			MotorPosChange_LeftIn:=ABS( Pos_LeftInMotor-Pos_LeftInMotor_Initial);
			IF MotorPosChange_LeftIn > Threshold_LeftInMotorPos THEN
				Alarm_LeftInMotorPos:=TRUE;
				ErrorID:=5009;
				ErrorDescription:='5009';
				Error:=TRUE;
				FB_PlcEmergencyStop();
				LED_Error:=TRUE;
			ELSE
				Alarm_LeftInMotorPos:=FALSE;
			END_IF
			//电机速度监测
			IF Velo_LeftInMotor > Threshold_LeftInMotorVelo THEN
				Alarm_LeftInMotorVelo:=TRUE;
				ErrorID:=5010;
				ErrorDescription:='5010';
				Error:=TRUE;
				FB_PlcEmergencyStop();
				LED_Error:=TRUE;
			ELSE
				Alarm_LeftInMotorVelo:=FALSE;
			END_IF
    ELSE
        Alarm_LeftInLin := FALSE;
	END_IF
END_IF
//RightIn monitor
IF DeltaVelo_RightInLin > LEHeartBeatDeadZone THEN
    // 有变动，光栅正常，计数器归零，更新位置,重置所有状态
    StableTimer_RightInLin(IN := FALSE, PT := LEHeartBeatAlarmTime);
    Alarm_RightInLin := FALSE;
    Velo_RightInLin_Last := RightInLin.NcToPlc.ActVelo;  // 
    StableTime_RightInLin := T#0S;
	IsInitialPositionSet_RightIn:=FALSE;
	Alarm_RightInMotorPos:=FALSE;
	Alarm_RightInMotorVelo:=FALSE;
ELSE
    //一点变动没有了，光栅异常，开始计时
    StableTimer_RightInLin(
        IN := TRUE,
        PT :=LEHeartBeatAlarmTime,
        ET => StableTime_RightInLin
    );
	//记录电机初始位置，后后续对比做准备
	IF NOT IsInitialPositionSet_RightIn THEN
        Pos_RightInMotor_Initial := Pos_RightInMotor;  // 记录初始位置
        IsInitialPositionSet_RightIn := TRUE;
   	END_IF;
    
    // 100ms速度完全不变，开始监控电机速度和位置
    IF StableTimer_RightInLin.Q THEN
        Alarm_RightInLin := TRUE;  // 
			//电机位置对比及监测
			MotorPosChange_RightIn:=ABS( Pos_RightInMotor-Pos_RightInMotor_Initial);
			IF MotorPosChange_RightIn > Threshold_RightInMotorPos THEN
				Alarm_RightInMotorPos:=TRUE;
				ErrorID:=5011;
				ErrorDescription:='5011';
				Error:=TRUE;
				FB_PlcEmergencyStop();
				LED_Error:=TRUE;
			ELSE
				Alarm_RightInMotorPos:=FALSE;
			END_IF
			//电机速度监测
			IF Velo_RightInMotor > Threshold_RightInMotorVelo THEN
				Alarm_RightInMotorVelo:=TRUE;
				ErrorID:=5012;
				ErrorDescription:='5012';
				Error:=TRUE;
				FB_PlcEmergencyStop();
				LED_Error:=TRUE;
			ELSE
				Alarm_RightInMotorVelo:=FALSE;
			END_IF
    ELSE
        Alarm_RightInLin := FALSE;
	END_IF
END_IF
//LeftOut monitor
IF DeltaVelo_LeftOutLin > LEHeartBeatDeadZone THEN
    // 有变动，光栅正常，计数器归零，更新位置,重置所有状态
    StableTimer_LeftOutLin(IN := FALSE, PT := LEHeartBeatAlarmTime);
    Alarm_LeftOutLin := FALSE;
    Velo_LeftOutLin_Last := LeftOutLin.NcToPlc.ActVelo;  // 
    StableTime_LeftOutLin := T#0S;
	IsInitialPositionSet_LeftOut:=FALSE;
	Alarm_LeftOutMotorPos:=FALSE;
	Alarm_LeftOutMotorVelo:=FALSE;
ELSE
    //一点变动没有了，光栅异常，开始计时
    StableTimer_LeftOutLin(
        IN := TRUE,
        PT := LEHeartBeatAlarmTime,
        ET => StableTime_LeftOutLin
    );
	//记录电机初始位置，后后续对比做准备
	IF NOT IsInitialPositionSet_LeftOut THEN
        Pos_LeftOutMotor_Initial := Pos_LeftOutMotor;  // 记录初始位置
        IsInitialPositionSet_LeftOut := TRUE;
   	END_IF;
    
    // 100ms速度完全不变，开始监控电机速度和位置
    IF StableTimer_LeftOutLin.Q THEN
        Alarm_LeftOutLin := TRUE;  // 
			//电机位置对比及监测
			MotorPosChange_LeftOut:=ABS( Pos_LeftOutMotor-Pos_LeftOutMotor_Initial);
			IF MotorPosChange_LeftOut > Threshold_LeftOutMotorPos THEN
				Alarm_LeftOutMotorPos:=TRUE;
				ErrorID:=5013;
				ErrorDescription:='5013';
				Error:=TRUE;
				FB_PlcEmergencyStop();
				LED_Error:=TRUE;
			ELSE
				Alarm_LeftOutMotorPos:=FALSE;
			END_IF
			//电机速度监测
			IF Velo_LeftOutMotor > Threshold_LeftOutMotorVelo THEN
				Alarm_LeftOutMotorVelo:=TRUE;
				ErrorID:=5014;
				ErrorDescription:='5014';
				Error:=TRUE;
				FB_PlcEmergencyStop();
				LED_Error:=TRUE;
			ELSE
				Alarm_LeftOutMotorVelo:=FALSE;
			END_IF
    ELSE
        Alarm_LeftOutLin := FALSE;
	END_IF
END_IF
//RightOut monitor
IF DeltaVelo_RightOutLin > LEHeartBeatDeadZone THEN
    // 有变动，光栅正常，计数器归零，更新位置,重置所有状态
    StableTimer_RightOutLin(IN := FALSE, PT := LEHeartBeatAlarmTime);
    Alarm_RightOutLin := FALSE;
    Velo_RightOutLin_Last := RightOutLin.NcToPlc.ActVelo;  // 
    StableTime_RightOutLin := T#0S;
	IsInitialPositionSet_RightOut:=FALSE;
	Alarm_RightOutMotorPos:=FALSE;
	Alarm_RightOutMotorVelo:=FALSE;
ELSE
    //一点变动没有了，光栅异常，开始计时
    StableTimer_RightOutLin(
        IN := TRUE,
        PT := LEHeartBeatAlarmTime,
        ET => StableTime_RightOutLin
    );
	//记录电机初始位置，后后续对比做准备
	IF NOT IsInitialPositionSet_RightOut THEN
        Pos_RightOutMotor_Initial := Pos_RightOutMotor;  // 记录初始位置
        IsInitialPositionSet_RightOut := TRUE;
   	END_IF;
    
    // 100ms速度完全不变，开始监控电机速度和位置
    IF StableTimer_RightOutLin.Q THEN
        Alarm_RightOutLin := TRUE;  // 
			//电机位置对比及监测
			MotorPosChange_RightOut:=ABS( Pos_RightOutMotor-Pos_RightOutMotor_Initial);
			IF MotorPosChange_RightOut > Threshold_RightOutMotorPos THEN
				Alarm_RightOutMotorPos:=TRUE;
				ErrorID:=5015;
				ErrorDescription:='5015';
				Error:=TRUE;
				FB_PlcEmergencyStop();
				LED_Error:=TRUE;
			ELSE
				Alarm_RightOutMotorPos:=FALSE;
			END_IF
			//电机速度监测
			IF Velo_RightOutMotor > Threshold_RightOutMotorVelo THEN
				Alarm_RightOutMotorVelo:=TRUE;
				ErrorID:=5016;
				ErrorDescription:='5016';
				Error:=TRUE;
				FB_PlcEmergencyStop();
				LED_Error:=TRUE;
			ELSE
				Alarm_RightOutMotorVelo:=FALSE;
			END_IF
    ELSE
        Alarm_RightOutLin := FALSE;
	END_IF
END_IF
END_ACTION

ACTION A_LoadOpcIocShellExe:
R_TRIG_Exeload(CLK:=bExe_load_Prog, Q=> );
LoadOpcIocTON(PT:=T#10S);
CASE Exe_load_step OF
	0:
		LoadOpcIocTON.IN:=TRUE;
		IF R_TRIG_Exeload.Q THEN
			NT_StartProcess_Load.START:=FALSE;
			NT_StartProcess_Load.PATHSTR:='C:\HZB\OpcIocShell\IDControlIOC\startTwinCATOPCServer.bat';
			Exe_load_step:=10;
		END_IF;
	10:
		IF LoadOpcIocTON.Q THEN
			NT_StartProcess_Load.START:=TRUE;
			Exe_load_step:=20;
		END_IF
	20:
		LoadOpcIocTON.IN:=FALSE;
		IF NT_StartProcess_Load.ERR THEN
			Exe_load_step:=0;
		ELSE
			Exe_load_step:=30;
		END_IF;
	30:
		IF NOT NT_StartProcess_Load.BUSY THEN
			NT_StartProcess_Load.START:=FALSE;
			Exe_Load_Done:=TRUE;
			Exe_load_step:=0;
		END_IF;
END_CASE;

NT_StartProcess_Load(
	NETID:='' ,
	PATHSTR:= ,
	DIRNAME:= , 
	COMNDLINE:= , 
	START:= ,
	ERRID=> );
END_ACTION

ACTION A_MonitorMotorAndLE:
//Monitoring Motor and LE Position/Velocity
IF 	ABS(DeltaPos_LeftTop) > ThresholdDeltaPos_LeftTop THEN
	ErrorID:=6001;
	Error:=TRUE;
	ErrorDescription:='ABS(DeltaPos_LeftTop) > ThresholdDeltaPos_LeftTop';
	FB_PlcEmergencyStop();
	LED_Error:=TRUE;
END_IF
IF ABS(DeltaPos_RightTop) > ThresholdDeltaPos_RightTop THEN
	ErrorID:=6002;
	Error:=TRUE;
	ErrorDescription:='ABS(DeltaPos_RightTop) > ThresholdDeltaPos_RightTop';
	FB_PlcEmergencyStop();
	LED_Error:=TRUE;
END_IF
IF ABS(DeltaPos_LeftBottom) > ThresholdDeltaPos_LeftBottom THEN
	ErrorID:=6003;
	Error:=TRUE;
	ErrorDescription:='ABS(DeltaPos_LeftBottom) > ThresholdDeltaPos_LeftBottom';
	FB_PlcEmergencyStop();
	LED_Error:=TRUE;
END_IF
IF ABS(DeltaPos_RightBottom) > ThresholdDeltaPos_RightBottom THEN
	ErrorID:=6004;
	Error:=TRUE;
	ErrorDescription:='ABS(DeltaPos_RightBottom) > ThresholdDeltaPos_RightBottom';
	FB_PlcEmergencyStop();
	LED_Error:=TRUE;
END_IF
IF 	ABS(DeltaPos_LeftIn) > ThresholdDeltaPos_LeftIn THEN
	ErrorID:=6001;
	Error:=TRUE;
	ErrorDescription:='ABS(DeltaPos_LeftIn) > ThresholdDeltaPos_LeftIn';
	FB_PlcEmergencyStop();
	LED_Error:=TRUE;
END_IF
IF ABS(DeltaPos_RightIn) > ThresholdDeltaPos_RightIn THEN
	ErrorID:=6002;
	Error:=TRUE;
	ErrorDescription:='ABS(DeltaPos_RightIn) > ThresholdDeltaPos_RightIn';
	FB_PlcEmergencyStop();
	LED_Error:=TRUE;
END_IF
IF ABS(DeltaPos_LeftOut) > ThresholdDeltaPos_LeftOut THEN
	ErrorID:=6003;
	Error:=TRUE;
	ErrorDescription:='ABS(DeltaPos_LeftOut) > ThresholdDeltaPos_LeftOut';
	FB_PlcEmergencyStop();
	LED_Error:=TRUE;
END_IF
IF ABS(DeltaPos_RightOut) > ThresholdDeltaPos_RightOut THEN
	ErrorID:=6004;
	Error:=TRUE;
	ErrorDescription:='ABS(DeltaPos_RightOut) > ThresholdDeltaPos_RightOut';
	FB_PlcEmergencyStop();
	LED_Error:=TRUE;
END_IF


IF ABS(DeltaVelo_LeftTop) > ThresholdDeltaVelo_LeftTop THEN
	ErrorID:=6005;
	Error:=TRUE;
	ErrorDescription:='ABS(DeltaVelo_LeftTop) > ThresholdDeltaVelo_LeftTop';
	FB_PlcEmergencyStop();
	LED_Error:=TRUE;
END_IF
IF ABS(DeltaVelo_RightTop) > ThresholdDeltaVelo_RightTop THEN
	ErrorID:=6006;
	Error:=TRUE;
	ErrorDescription:='ABS(DeltaVelo_RightTop) > ThresholdDeltaVelo_RightTop';
	FB_PlcEmergencyStop();
	LED_Error:=TRUE;
END_IF
IF ABS(DeltaVelo_LeftBottom) > ThresholdDeltaVelo_LeftBottom THEN
	ErrorID:=6007;
	Error:=TRUE;
	ErrorDescription:='ABS(DeltaVelo_LeftBottom) > ThresholdDeltaVelo_LeftBottom';
	FB_PlcEmergencyStop();
	LED_Error:=TRUE;
END_IF
IF ABS(DeltaVelo_RightBottom) > ThresholdDeltaVelo_RightBottom THEN
	ErrorID:=6008;
	Error:=TRUE;
	ErrorDescription:='ABS(DeltaVelo_RightBottom) > ThresholdDeltaVelo_RightBottom';
	FB_PlcEmergencyStop();
	LED_Error:=TRUE;
END_IF
IF ABS(DeltaVelo_LeftIn) > ThresholdDeltaVelo_LeftIn THEN
	ErrorID:=6005;
	Error:=TRUE;
	ErrorDescription:='ABS(DeltaVelo_LeftIn) > ThresholdDeltaVelo_LeftIn';
	FB_PlcEmergencyStop();
	LED_Error:=TRUE;
END_IF
IF ABS(DeltaVelo_RightIn) > ThresholdDeltaVelo_RightIn THEN
	ErrorID:=6006;
	Error:=TRUE;
	ErrorDescription:='ABS(DeltaVelo_RightIn) > ThresholdDeltaVelo_RightIn';
	FB_PlcEmergencyStop();
	LED_Error:=TRUE;
END_IF
IF ABS(DeltaVelo_LeftOut) > ThresholdDeltaVelo_LeftOut THEN
	ErrorID:=6007;
	Error:=TRUE;
	ErrorDescription:='ABS(DeltaVelo_LeftOut) > ThresholdDeltaVelo_LeftOut';
	FB_PlcEmergencyStop();
	LED_Error:=TRUE;
END_IF
IF ABS(DeltaVelo_RightOut) > ThresholdDeltaVelo_RightOut THEN
	ErrorID:=6008;
	Error:=TRUE;
	ErrorDescription:='ABS(DeltaVelo_RightOut) > ThresholdDeltaVelo_RightOut';
	FB_PlcEmergencyStop();
	LED_Error:=TRUE;
END_IF
(*
//
//IF NotMoving ,Threshold is less
//
IF NOT moveStatusLeftTop THEN
		IF 	ABS(DeltaPos_LeftTop) > ThresholdDeltaPos_LeftTop/3 THEN
		ErrorID:=6009;
		Error:=TRUE;
		ErrorDescription:='ABS(DeltaPos_LeftTop) > ThresholdDeltaPos_LeftTop/3';
		FB_PlcEmergencyStop();
		LED_Error:=TRUE;
	END_IF
END_IF
IF NOT moveStatusRightTop THEN
	IF ABS(DeltaPos_RightTop) > ThresholdDeltaPos_RightTop/3 THEN
		ErrorID:=6010;
		Error:=TRUE;
		ErrorDescription:='ABS(DeltaPos_RightTop) > ThresholdDeltaPos_RightTop/3';
		FB_PlcEmergencyStop();
		LED_Error:=TRUE;
	END_IF
END_IF
IF NOT moveStatusLeftBottom THEN
	IF ABS(DeltaPos_LeftBottom) > ThresholdDeltaPos_LeftBottom/3 THEN
		ErrorID:=6011;
		Error:=TRUE;
		ErrorDescription:='ABS(DeltaPos_LeftBottom) > ThresholdDeltaPos_LeftBottom/3';
		FB_PlcEmergencyStop();
		LED_Error:=TRUE;
	END_IF
END_IF
IF NOT moveStatusRightBottom THEN
	IF ABS(DeltaPos_RightBottom) > ThresholdDeltaPos_RightBottom/3 THEN
		ErrorID:=6012;
		Error:=TRUE;
		ErrorDescription:='ABS(DeltaPos_RightBottom) > ThresholdDeltaPos_RightBottom';
		FB_PlcEmergencyStop();
		LED_Error:=TRUE;
	END_IF
END_IF

//
IF NOT moveStatusLeftTop THEN
	IF ABS(DeltaVelo_LeftTop) > ThresholdDeltaVelo_LeftTop/3 THEN
		ErrorID:=6013;
		Error:=TRUE;
		ErrorDescription:='ABS(DeltaVelo_LeftTop) > ThresholdDeltaVelo_LeftTop/3';
		FB_PlcEmergencyStop();
		LED_Error:=TRUE;
	END_IF
END_IF
IF NOT moveStatusRightTop THEN
	IF ABS(DeltaVelo_RightTop) > ThresholdDeltaVelo_RightTop/3 THEN
		ErrorID:=6014;
		Error:=TRUE;
		ErrorDescription:='ABS(DeltaVelo_RightTop) > ThresholdDeltaVelo_RightTop/3';
		FB_PlcEmergencyStop();
		LED_Error:=TRUE;
	END_IF
END_IF
IF NOT moveStatusLeftBottom THEN
	IF ABS(DeltaVelo_LeftBottom) > ThresholdDeltaVelo_LeftBottom/3 THEN
		ErrorID:=6015;
		Error:=TRUE;
		ErrorDescription:='ABS(DeltaVelo_LeftBottom) > ThresholdDeltaVelo_LeftBottom/3';
		FB_PlcEmergencyStop();
		LED_Error:=TRUE;
	END_IF
END_IF
IF NOT moveStatusRightBottom THEN
	IF ABS(DeltaVelo_RightBottom) > ThresholdDeltaVelo_RightBottom/3 THEN
		ErrorID:=6016;
		Error:=TRUE;
		ErrorDescription:='ABS(DeltaVelo_RightBottom) > ThresholdDeltaVelo_RightBottom/3';
		FB_PlcEmergencyStop();
		LED_Error:=TRUE;
	END_IF
END_IF
*)
END_ACTION

ACTION A_PosDiffDetectiion:
IF ABS(PosDiff_LeftTopLin_actual)>PosDiff_LeftTopLin THEN
	ErrorID:=201;
	Error:=TRUE;
	ErrorDescription:='ABS(PosDiff_LeftTopLin_actual)>PosDiff_LeftTopLin';
	FB_PlcEmergencyStop();
	LED_Error:=TRUE;
END_IF
IF ABS(PosDiff_RightTopLin_actual)>PosDiff_RightTopLin THEN
	ErrorID:=202;
	Error:=TRUE;
	ErrorDescription:='ABS(PosDiff_RightTopLin_actual)>PosDiff_RightTopLin';
	FB_PlcEmergencyStop();
	LED_Error:=TRUE;
END_IF
IF ABS(PosDiff_LeftBottomLin_actual)>PosDiff_LeftBottomLin THEN
	ErrorID:=203;
	Error:=TRUE;
	ErrorDescription:='ABS(PosDiff_LeftBottomLin_actual)>PosDiff_LeftBottomLin';
	FB_PlcEmergencyStop();
	LED_Error:=TRUE;
END_IF
IF ABS(PosDiff_RightBottomLin_actual)>PosDiff_RightBottomLin THEN
	ErrorID:=204;
	ErrorDescription:='ABS(PosDiff_RightBottomLin_actual)>PosDiff_RightBottomLin';
	Error:=TRUE;
	FB_PlcEmergencyStop();
	LED_Error:=TRUE;
END_IF
//
IF ABS(PosDiff_LeftTopLin_actual-PosDiff_RightTopLin_actual)>0.05 THEN
	ErrorID:=205;
	ErrorDescription:='ABS(PosDiff_LeftTopLin_actual-PosDiff_RightTopLin_actual)>0.05';
	Error:=TRUE;
	FB_PlcEmergencyStop();
	LED_Error:=TRUE;
ELSIF ABS(PosDiff_LeftBottomLin_actual-PosDiff_RightBottomLin_actual)>0.05 THEN
	ErrorID:=206;
	ErrorDescription:='ABS(PosDiff_LeftBottomLin_actual-PosDiff_RightBottomLin_actual)>0.05';
	Error:=TRUE;
	FB_PlcEmergencyStop();
	LED_Error:=TRUE;
END_IF

//In out
IF ABS(PosDiff_LeftInLin_actual)>PosDiff_LeftInLin THEN
	ErrorID:=201;
	Error:=TRUE;
	ErrorDescription:='ABS(PosDiff_LeftInLin_actual)>PosDiff_LeftInLin';
	FB_PlcEmergencyStop();
	LED_Error:=TRUE;
END_IF
IF ABS(PosDiff_RightInLin_actual)>PosDiff_RightInLin THEN
	ErrorID:=202;
	Error:=TRUE;
	ErrorDescription:='ABS(PosDiff_RightInLin_actual)>PosDiff_RightInLin';
	FB_PlcEmergencyStop();
	LED_Error:=TRUE;
END_IF
IF ABS(PosDiff_LeftOutLin_actual)>PosDiff_LeftOutLin THEN
	ErrorID:=203;
	Error:=TRUE;
	ErrorDescription:='ABS(PosDiff_LeftOutLin_actual)>PosDiff_LeftOutLin';
	FB_PlcEmergencyStop();
	LED_Error:=TRUE;
END_IF
IF ABS(PosDiff_RightOutLin_actual)>PosDiff_RightOutLin THEN
	ErrorID:=204;
	ErrorDescription:='ABS(PosDiff_RightOutLin_actual)>PosDiff_RightOutLin';
	Error:=TRUE;
	FB_PlcEmergencyStop();
	LED_Error:=TRUE;
END_IF
//
IF ABS(PosDiff_LeftTopLin_actual-PosDiff_RightTopLin_actual)>0.05 THEN
	ErrorID:=205;
	ErrorDescription:='ABS(PosDiff_LeftTopLin_actual-PosDiff_RightTopLin_actual)>0.05';
	Error:=TRUE;
	FB_PlcEmergencyStop();
	LED_Error:=TRUE;
ELSIF ABS(PosDiff_LeftOutLin_actual-PosDiff_RightOutLin_actual)>0.05 THEN
	ErrorID:=206;
	ErrorDescription:='ABS(PosDiff_LeftOutLin_actual-PosDiff_RightOutLin_actual)>0.05';
	Error:=TRUE;
	FB_PlcEmergencyStop();
	LED_Error:=TRUE;
END_IF
END_ACTION

ACTION A_RestartDrivers:
Relay_EL2624[0]:=btn_RestartDriver1;
Relay_EL2624[1]:=btn_RestartDriver2;
Relay_EL2624[2]:=btn_RestartDriver3;
Relay_EL2624[3]:=btn_RestartDriver4;
Relay_EL2624[4]:=btn_RestartDriver5;
Relay_EL2624[5]:=btn_RestartDriver6;
Relay_EL2624[6]:=btn_RestartDriver7;
Relay_EL2624[7]:=btn_RestartDriver8;
///
//1.上升沿触发，btn_RestartDrivers上升沿后，btn_RestartDriver1~8全部高电平
//2、3s后，Driver1~8全部恢复低电平
//3、恢复全部状态到初始
///
RestartDriver_RTRIG(CLK:=btn_RestartDriversAll);
IF RestartDriver_RTRIG.Q THEN
	RestartDriver_Triggered:=TRUE;
	RestartDriver_Done:=FALSE;
END_IF
IF RestartDriver_Triggered THEN
	CASE RestartDriver_State OF
		0:
			btn_RestartDriver1:=TRUE;
			btn_RestartDriver2:=TRUE;
			btn_RestartDriver3:=TRUE;
			btn_RestartDriver4:=TRUE;
			btn_RestartDriver5:=TRUE;
			btn_RestartDriver6:=TRUE;
			btn_RestartDriver7:=TRUE;
			btn_RestartDriver8:=TRUE;
			//计时开始
			RestartDriver_TON(PT:=T#10S);
			RestartDriver_TON.IN:=TRUE;
			IF RestartDriver_TON.Q THEN
				RestartDriver_State:=1;
			END_IF
		1:
			btn_RestartDriver1:=FALSE;
			btn_RestartDriver2:=FALSE;
			btn_RestartDriver3:=FALSE;
			btn_RestartDriver4:=FALSE;
			btn_RestartDriver5:=FALSE;
			btn_RestartDriver6:=FALSE;
			btn_RestartDriver7:=FALSE;
			btn_RestartDriver8:=FALSE;
			RestartDriver_State:=88;
		88:
			RestartDriver_TON.IN:=FALSE;
			btn_RestartDriversAll:=FALSE;
			RestartDriver_State:=0;
			RestartDriver_Triggered:=FALSE;
			RestartDriver_Done:=TRUE;
	END_CASE
END_IF
END_ACTION

ACTION A_RestartTC:
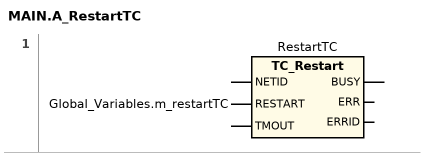
// NETWORK 1
RestartTC(RESTART := Global_Variables.m_restartTC); // TC_Restart
END_ACTION

ACTION A_SafePlcStartInit:
fb_ton0(PT:=t#1s);
fb_ton1(PT:=t#0.1s);
fb_ton2(PT:=t#0.1s);
fb_ton3(PT:=t#0.1s);

CASE SafeStatus OF
	0:
		IF COM_ERROR OR NOT Estop_Out THEN
			Err_Ack:=TRUE;
			fb_ton0.IN:=TRUE;
			SafeStatus:=1;
		ELSE
			SafePLCRunOK:=TRUE;
			SafeStatus:=0;
		END_IF
	1:
		IF fb_ton0.Q THEN
			Err_Ack:=FALSE;
			Safe_run:=TRUE;
			fb_ton1.IN:=TRUE;
			SafeStatus:=2;
		END_IF

	2:
		IF fb_ton1.Q THEN
			IF Estop_RunAndRestart=FALSE THEN
				Estop_RunAndRestart:=TRUE;
				fb_ton2.IN:=TRUE;
				SafeStatus:=3;
			END_IF
		END_IF
	3:
		IF fb_ton2.Q THEN
			IF Estop_RunAndRestart THEN
				Estop_RunAndRestart:=FALSE;
				fb_ton3.IN:=TRUE;
				SafeStatus:=4;
			END_IF
		END_IF
	4:
		IF fb_ton3.Q THEN
			IF Estop_Out THEN
				SafePLCRunOK:=TRUE;
				SafeStatus:=0;
			ELSE
				SafePLCRunOK:=FALSE;
				//Error:=TRUE;
				//ErrorId:=301;
				//ErrorDescription:='SafePLCRunOK fail';
			END_IF
		fb_ton0.IN:=FALSE;
		fb_ton1.IN:=FALSE;
		fb_ton2.IN:=FALSE;
		fb_ton3.IN:=FALSE;
		END_IF


END_CASE
END_ACTION

ACTION A_SetAxisPosition:
fb_ton4(PT:=t#0.5s);
CASE SetAxisPosState OF
	0:	(*FB_Set_AxisPosition*)
		FB_Set_AxisPosition(Execute:=TRUE);
		fb_ton4.IN:=TRUE;
		SetAxisPosState:=1;
	1:	(*wait*)
		FB_Set_AxisPosition();
		IF NOT FB_Set_AxisPosition.Done THEN		(*FB_Set_AxisPositionÃ»ÓÐÖ´ÐÐÍê£¬wait£¬³¬Ê±FB Error*)
			IF NOT fb_ton4.Q THEN
				SetAxisPosState:=1;
			ELSE
				SetAxisPosState:=99;
			END_IF
		ELSE
			SetAxisPosState:=88;
		END_IF
	88:
		SetAxisPosState:=0;
		SerAxisPositionDone:=TRUE;
		Error:=FALSE;
		ErrorID:=0;
		FB_Set_AxisPosition.Execute:=FALSE;
		fb_ton4.IN:=FALSE;
	99:
		SetAxisPosState:=99;
		SerAxisPositionDone:=FALSE;
		Error:=TRUE;
		FB_Set_AxisPosition.Execute:=FALSE;
		fb_ton4.IN:=FALSE;
		LED_Error:=TRUE;
		ErrorID:=401;
		ErrorDescription:='SetAxisPosition fail';
END_CASE
END_ACTION

ACTION A_SetLinearEncoderPositionBias:
//光栅positionBias补偿低温收缩量
//IF CryogenicCompensationConditionsReady AND NOT CryogenicCompensationDone THEN
//	PositionBias_LeftTop:=PositionBias_LeftTop+CryogenicCompensation_LeftTop;
//	PositionBias_RightTop:=PositionBias_RightTop+CryogenicCompensation_RightTop;
//	PositionBias_LeftBottom:=PositionBias_LeftBottom+CryogenicCompensation_LeftBottom;
//	PositionBias_RightBottom:=PositionBias_RightBottom+CryogenicCompensation_RightBottom;
//	CryogenicCompensationDone:=TRUE;
//END_IF
//设置bias开始
A_SetLinearEncoderPositionBiasMC();
PositionBiasTON(PT:=T#0.1S);
CASE state_setLEPosBias OF
	0:
		PositionBiasTON.IN:=TRUE;
		IF MC_SetLEPosBias_LeftTop.Error OR MC_SetLEPosBias_RightTop.Error OR 
			MC_SetLEPosBias_LeftBottom.Error OR MC_SetLEPosBias_RightBottom.Error OR
			MC_SetLEPosBias_LeftIn.Error OR MC_SetLEPosBias_RightIn.Error OR 
			MC_SetLEPosBias_LeftOut.Error OR MC_SetLEPosBias_RightOut.Error THEN
			state_setLEPosBias:=-100;
		ELSE 
			state_setLEPosBias:=1;
		END_IF
	1:
		IF NOT MC_SetLEPosBias_LeftTop.Done OR NOT MC_SetLEPosBias_RightTop.Done OR 
			NOT MC_SetLEPosBias_LeftBottom.Done OR NOT MC_SetLEPosBias_RightBottom.Done OR
			NOT MC_SetLEPosBias_LeftIn.Done OR NOT MC_SetLEPosBias_RightIn.Done OR 
			NOT MC_SetLEPosBias_LeftOut.Done OR NOT MC_SetLEPosBias_RightOut.Done THEN
			MC_SetLEPosBias_LeftTop.Execute:=TRUE;
			MC_SetLEPosBias_RightTop.Execute:=TRUE;
			MC_SetLEPosBias_LeftBottom.Execute:=TRUE;
			MC_SetLEPosBias_RightBottom.Execute:=TRUE;
			MC_SetLEPosBias_LeftIn.Execute:=TRUE;
			MC_SetLEPosBias_RightIn.Execute:=TRUE;
			MC_SetLEPosBias_LeftOut.Execute:=TRUE;
			MC_SetLEPosBias_RightOut.Execute:=TRUE;
			state_setLEPosBias:=2;
		ELSE
			state_setLEPosBias:=-100;
		END_IF
	2:
		IF NOT MC_SetLEPosBias_LeftTop.Done OR NOT MC_SetLEPosBias_RightTop.Done OR 
			NOT MC_SetLEPosBias_LeftBottom.Done OR NOT MC_SetLEPosBias_RightBottom.Done OR
			NOT MC_SetLEPosBias_LeftIn.Done OR NOT MC_SetLEPosBias_RightIn.Done OR 
			NOT MC_SetLEPosBias_LeftOut.Done OR NOT MC_SetLEPosBias_RightOut.Done THEN
			IF NOT PositionBiasTON.Q THEN
				state_setLEPosBias:=2;
			ELSE
				state_setLEPosBias:=-100;
			END_IF
		END_IF
		IF  MC_SetLEPosBias_LeftTop.Done AND MC_SetLEPosBias_RightTop.Done AND
			MC_SetLEPosBias_LeftBottom.Done AND MC_SetLEPosBias_RightBottom.Done AND 
			MC_SetLEPosBias_LeftIn.Done AND MC_SetLEPosBias_RightIn.Done AND
			MC_SetLEPosBias_LeftOut.Done AND MC_SetLEPosBias_RightOut.Done THEN
			state_setLEPosBias:=88;
		END_IF	
		IF MC_SetLEPosBias_LeftTop.Error OR MC_SetLEPosBias_RightTop.Error OR 
			MC_SetLEPosBias_LeftBottom.Error OR MC_SetLEPosBias_RightBottom.Error OR 
			MC_SetLEPosBias_LeftIn.Error OR MC_SetLEPosBias_RightIn.Error OR 
			MC_SetLEPosBias_LeftOut.Error OR MC_SetLEPosBias_RightOut.Error THEN
			state_setLEPosBias:=-100;
		END_IF 
		
	88:
		PositionBiasTON.IN:=FALSE;
		PositionBiasDone:=TRUE;
	-100:
		PositionBiasTON.IN:=FALSE;
		PositionBiasDone:=FALSE;
		Error:=TRUE;
		ErrorId:=901;
		ErrorDescription:='Set LinearEncoderPositionBias Error';
		Plc_EmergencyStop:=FALSE;
END_CASE
END_ACTION

ACTION A_SetLinearEncoderPositionBiasMC:
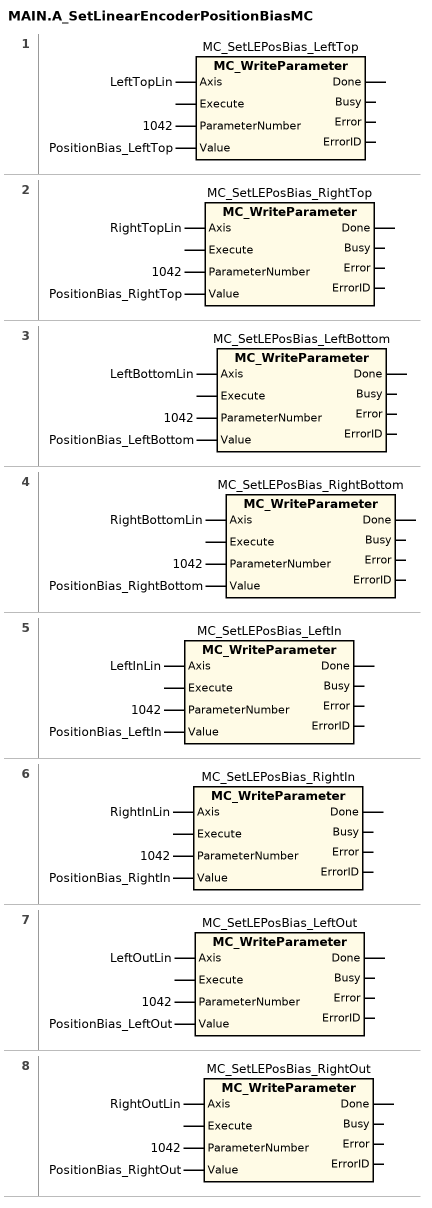
// NETWORK 1
MC_SetLEPosBias_LeftTop(Axis := LeftTopLin, ParameterNumber := 1042, Value := PositionBias_LeftTop); // MC_WriteParameter

// NETWORK 2
MC_SetLEPosBias_RightTop(Axis := RightTopLin, ParameterNumber := 1042, Value := PositionBias_RightTop); // MC_WriteParameter

// NETWORK 3
MC_SetLEPosBias_LeftBottom(Axis := LeftBottomLin, ParameterNumber := 1042, Value := PositionBias_LeftBottom); // MC_WriteParameter

